Omron CX-Programmer project NewProject (CX-Programmer 9.66)

# PLC LQK19011ICM: CP1H XA
I/O table (CPU CP1H-XA40DR-A): rack 0 slot 0 CJ1W-SCU21

## Global symbols (name address type ; comment)
AI_SAW_CURRENT 200 CHANNEL  ; ANALOG.INPUT1.SAW.CURRENT
AO_TRANS_VEL_REF 210 CHANNEL  ; TRANSVERSE.AXIS.VELOCITY.ANALOG.REFERENCE
0 CHANNEL  ; Zero Jog reference value first
0.04 BOOL  ; SPARE
0.05 BOOL  ; SPARE
1.01 BOOL  ; Spare
1.03 BOOL  ; Spare
D10 CHANNEL  ; Jog Velocity Reference Value
D1000 CHANNEL  ; First Dtata address of block table
D2000 CHANNEL  ; First Data Word of slab table
D8 CHANNEL  ; Interim Jog Storage Wd
D9 CHANNEL  ; Interim Storage word for Jog
H10.11 BOOL  ; MC.LONG.AXIS
H10.12 BOOL  ; MC.LONG.AXIS
H10.13 BOOL  ; MC.LONG.AXIS
H12.07 BOOL  ; MC.TRANSVERSE.AXIS
H12.08 BOOL  ; MC.TRANSVERSE.AXIS
H12.11 BOOL  ; MC.TRANSVERSE.AXIS
H12.12 BOOL  ; MC.TRANSVERSE.AXiS
H12.13 BOOL  ; MC.TRANSVERSE.AXIS
T0000 BOOL  ; Step 0 Timer Done
T0001 BOOL  ; Step 1 Timer Done
T0002 BOOL  ; Step 2 timer done
T0003 BOOL  ; Increment Slab Pulse Timer
T0004 BOOL  ; Slab Decrement Pulse Timer
T0005 BOOL  ; Block Increment Pulse Timer
T0006 BOOL  ; Block Decrement Pulse Timer
T0010 BOOL  ; Block Step 0 Timer
T0011 BOOL  ; Block Step 1 Timer
T0012 BOOL  ; Block Step 2 Timer
T0013 BOOL  ; Block Step 3 Timer
T0014 BOOL  ; Block Step 4 timer
T0015 BOOL  ; Block Step 5 Timer
T0016 BOOL  ; Block Step 6 Timer
W121.02 BOOL  ; Previous Block
W121.03 BOOL  ; Previous Slab of Current Block
W121.04 BOOL  ; Next Slab of current Block
W121.05 BOOL  ; Next Block Select
W121.06 BOOL  ; Write Current Block to Storage (HMI PB)
W121.07 BOOL  ; Clear Data
W12.00 BOOL  ; Slab Change Data Storage and Display Update Step 0
W12.01 BOOL  ; Step 1
W12.02 BOOL  ; Step 2
W12.03 BOOL  ; Step 3
W12.04 BOOL  ; Step 4
W12.05 BOOL  ; Step 5
W12.06 BOOL  ; Step 6
W12.15 BOOL  ; Loop Step Reset
W13.00 BOOL  ; Step 0 in Progress
W13.01 BOOL  ; Step 1 in Progress
W13.02 BOOL  ; Step 2 in Progress
W13.03 BOOL  ; Step 3 in Progress
W13.04 BOOL  ; Step 4 in Progress
W13.05 BOOL  ; Step 5 in Progress
W13.06 BOOL  ; Step 6 in Progress
W14.00 BOOL  ; Step 0 Done
W14.01 BOOL  ; Step 1 Done
W14.02 BOOL  ; Step 2 Done
W14.03 BOOL  ; Step 3 Done
W14.04 BOOL  ; Step 4 Done
W14.05 BOOL  ; Step 5 Done
W14.06 BOOL  ; Step 6 Done
W150 CHANNEL  ; Block Number Captured
W151 CHANNEL  ; Number of Words for Blocks
W152 CHANNEL  ; Slab Count Work Word for Block Pointer
W153 CHANNEL  ; Offset Calculate for Last Slab Count
W154 CHANNEL  ; Offset Mid Calc
W156 CHANNEL  ; Offset Calc'd
W158 CHANNEL  ; Slab Record Offset Interim
W15.00 BOOL  ; Block Change Data Storage and Display Update Step 0
W15.01 BOOL  ; Loop Step 1
W15.02 BOOL  ; Loop Step 2
W15.03 BOOL  ; Loop Step 3
W15.04 BOOL  ; Loop Step 4
W15.05 BOOL  ; Loop Step 5
W15.06 BOOL  ; Loop Step 6
W15.15 BOOL  ; Loop Step Reset
W160 CHANNEL  ; Slab Offset Result
W16.00 BOOL  ; Step 0 in Progress
W16.01 BOOL  ; Loop Step 1 in Progress
W16.02 BOOL  ; Loop Step 2 in Progress
W16.03 BOOL  ; Loop Step 3 in Progress
W16.04 BOOL  ; Loop Step 4 in Progress
W16.05 BOOL  ; Loop Step 5 in Progress
W16.06 BOOL  ; Loop Step 6 in Progress
W16.10 BOOL  ; Slab Data Read in Progress
W16.11 BOOL  ; Block Data Read in Progress
W17.00 BOOL  ; Step 0 Done
W17.01 BOOL  ; Loop Step 1 Done
W17.02 BOOL  ; Loop Step 2 Complete
W17.03 BOOL  ; Loop Sstep 3 Complete
W17.04 BOOL  ; Loop Step 4 Complete
W17.05 BOOL  ; Loop Step 5 Complete
W17.06 BOOL  ; Loop Step 6 Complete
W190 CHANNEL  ; Slab Pointer Offset Adjustment
W191 CHANNEL  ; Block 1 Slab Count Capture
W192 CHANNEL  ; Slab Offset Addition for This Block
W193 CHANNEL  ; Slab_ID_Raw
W194 CHANNEL  ; Slab Pointer Calculated
W195 CHANNEL  ; Slab Offset Previous
W196 CHANNEL  ; Slab_Offset_Constant_Calculated
W197 CHANNEL  ; Block_Selected_Base
W198 CHANNEL  ; Block Pointer Offset Calculated
W19.00 BOOL  ; Test Bit
W19.01 BOOL  ; Self Toggle
W200 CHANNEL  ; Block ID
W201 CHANNEL  ; Number Of Blocks
W202 CHANNEL  ; Current Block Height
W203 CHANNEL  ; Current Block Start Edge
W204 CHANNEL  ; Current Block Length
W205 CHANNEL  ; Current Block First Cut Location
W206 CHANNEL  ; Current Block SLab Count
W207 CHANNEL  ; Slab ID
W208 CHANNEL  ; Current Slab Size in inches
W209 CHANNEL  ; Current Slab Quantity to cut
W20.00 BOOL  ; Block Incremented Pulse - Lead
W20.01 BOOL  ; Block Decremented Pulse - Lead
W20.02 BOOL  ; Slab Incremented Pulse - Lead
W20.03 BOOL  ; Slab Decremented Pulse - Lead
W20.04 BOOL  ; Slab Count Capture Trap
W20.05 BOOL  ; Block Read In Progress
W20.06 BOOL  ; Slab Count Changed from Block Read
W20.07 BOOL  ; Slab Pointer Updating
W20.08 BOOL  ; Update Working Offset
W20.09 BOOL  ; Block Pointer Calculate Enable
W20.10 BOOL  ; Increment Block Pointer
W20.11 BOOL  ; Decrement Block Pointer
W20.12 BOOL  ; First_Pass_Read
W20.14 BOOL  ; Block Offset Calculated
W20.15 BOOL  ; Block Program Control Enabled
W21.00 BOOL  ; Blade Kerf Data Write to Storage
W21.01 BOOL  ; Blade Kerf Read from Storage
W21.02 BOOL  ; Cut Depth Write to Storage
W21.03 BOOL  ; Cut Depth Read from Storage
W21.04 BOOL  ; Target Saw Current in Amps Write to Storage
W21.05 BOOL  ; Target Saw Current in Amps Read from Storage
W21.06 BOOL  ; Read Slab Data from Storage
W21.07 BOOL  ; Block Data Write to Storage
W21.08 BOOL  ; Automatic Number of Blocks Update
W21.09 BOOL  ; Slab Pointer Control Enabled
W21.10 BOOL  ; Increment Slab Offset
W21.11 BOOL  ; Decrement Slab Offset
W21.12 BOOL  ; Automatic Number of Slabs Update
W21.13 BOOL  ; Slab Pointer Reset
W21.14 BOOL  ; Block Pointer Reset
W22.00 BOOL  ; Slab Pointer Calculated
W22.01 BOOL  ; Block Pointer Changed
W22.02 BOOL  ; Current Block Selected Changed Initiate Block Data Write
W22.03 BOOL  ; Block Data Write Step Zero Complete
W22.04 BOOL  ; Block Data Write Complete
W22.05 BOOL  ; Capture Current Slab Words
W22.06 BOOL  ; Slab Data Write In Progress
W22.07 BOOL  ; Slab Data Write Complete
W22.08 BOOL  ; Block Offset Adjusted
W22.09 BOOL  ; Block Offset Adjust Complete
W22.10 BOOL  ; Block Data Read in Progress
W22.11 BOOL  ; Block Data Read >
W22.12 BOOL  ; Block Data Read Complete
W22.13 BOOL  ; Slab Offset Adjust in Progress
W22.14 BOOL  ; Slab Offset Adjust >
W22.15 BOOL  ; Slab Offset Adjust Complete
W23.00 BOOL  ; Slab Offset Init
W23.01 BOOL  ; Slab Offset Pointer Updating
W23.02 BOOL  ; Slab Offset Updated
W23.03 BOOL  ; Slab Data Read in Progress
W23.04 BOOL  ; Slab Data Read >
W23.05 BOOL  ; Slab Data Read Complete
W23.15 BOOL  ; Slab Offset Init Complete
W24.01 BOOL  ; Offset Init Step 1 Complete
W24.02 BOOL  ; OffsetInit Step 2 Complete
W24.03 BOOL  ; Offset Init Step 3 Complete
W250 CHANNEL  ; Offset value for Second word in indirect addressed storage area for Block Start Edge
W251 CHANNEL  ; Offset Value for Third word in Storge area for block length
W252 CHANNEL  ; Offset value calculated for 4th word in Storage area for block First Cut
W253 CHANNEL  ; Offset value calculated for number of slabs for current block
W256 CHANNEL  ; Last Slab Count from First Block
W257 CHANNEL  ; Offset adjust
W25.01 BOOL  ; Offset Init Step 1 In Progress
W25.02 BOOL  ; Offset Init Step 2 In Progress
W25.03 BOOL  ; Offset Init Step 3 In Progress
W26.00 BOOL  ; Minus Slab Offset Init
W26.01 BOOL  ; Minus Offset Init Step 1
W26.02 BOOL  ; Minus Offset Init Step 2
W26.03 BOOL  ; Minus Offset Init Step 3
W26.15 BOOL  ; Minus Slab Offset Init Complete
W27.01 BOOL  ; Minus Offset Init Step 1 Complete
W27.02 BOOL  ; Minus Offset Init Step 2 Complete
W27.03 BOOL  ; Minus Offset Init Step 3 Complete
W28.01 BOOL  ; Minus Offset Init Step 1 In Progress
W28.02 BOOL  ; Minus Offset Init Step 2 In Progress
W28.03 BOOL  ; Minus Offset Init Step 3 In Progress
W300 CHANNEL  ; Blade Kerf Working
W301 CHANNEL  ; Cut Depth Working
W302 CHANNEL  ; Target Current Working
W30.00 BOOL  ; OI.MESSAGE.INTERNAL.TRIGGER.MSG0
W30.01 BOOL  ; OI.MESSAGE.INTERNAL.TRIGGER.MSG1
W312 CHANNEL  ; Last Height Value for Current Block
W313 CHANNEL  ; Current Block Stored Height Data
W314 CHANNEL  ; Curren Block Last Start Edge
W315 CHANNEL  ; Current Block Stored Start Edge
W316 CHANNEL  ; Current Block Last Length
W317 CHANNEL  ; Current Block Stored Length
W318 CHANNEL  ; Current Block Last First Cut Position
W319 CHANNEL  ; Current Block Stored First Cut Location
W320 CHANNEL  ; Current Block Last Number of Slabs
W321 CHANNEL  ; Current Block Stored Slab Count
W322 CHANNEL  ; Current Slab Last Width
W323 CHANNEL  ; Current Slab Stored Width
W324 CHANNEL  ; Current Slab Last Quantity
W325 CHANNEL  ; Current Slab Stored Quantity
W37.00 BOOL  ; Current Height and Last Height are not Equal after Block Inc/Dec
W37.01 BOOL  ; Last Height and Stored Height are not Equal
W37.02 BOOL  ; Current Block Start Edge and Last Block Start Edge are Not Equal
W37.03 BOOL  ; Last Block Start Edge and Stored Value are Not Equal
W37.04 BOOL  ; Current Block Length and Last Block Length are Not Equal
W37.05 BOOL  ; Last Block Length and Stored Length are Not Equal
W37.06 BOOL  ; Current and Last First Cut Location are Not Equal
W37.07 BOOL  ; Last and Stored First Cut Location are Not Equal
W37.08 BOOL  ; Last and Current Slab Count are Not Equal
W37.09 BOOL  ; Last and Stored Slab Count are Not Equal
W37.10 BOOL  ; Current and Last Slab Size are Not Equal
W37.11 BOOL  ; Last and Stored Slab Sizes are Not Equal
W37.12 BOOL  ; Last and Current Slab Qty are Not Equal
W37.13 BOOL  ; Last and Stored Slab Qty are Not Equal
W400 CHANNEL  ; Temporary Storage for Block Data Used in Slab Offset Calc
W400.00 BOOL  ; Data Write Step
W400.01 BOOL  ; Data Offset Adjust Step
W400.02 BOOL  ; Data Read Step
W400.03 BOOL  ; End Step
W404 CHANNEL  ; # of Slabs for current Block
W405 CHANNEL  ; Number of words used by slabs in this block
W406 CHANNEL  ; Temporary Offset Storage word
W40.00 BOOL  ; Data Write/Read Sequence Initiate
W40.01 BOOL  ; Data Write Step Action
W40.02 BOOL  ; Data Offset Adjust Action
W40.03 BOOL  ; Data Read Step Action
W41.00 BOOL  ; Slab Data Write in Progress
W41.01 BOOL  ; Slab Data Write >
W41.02 BOOL  ; Slab Offset Adjust in Progress
W41.03 BOOL  ; Calulating Number of Words to Read
W90.00 BOOL  ; Block Data Write Step 0
W90.01 BOOL  ; Slab Data Write Step 1
W90.02 BOOL  ; Change Block Offset Pointer
W90.03 BOOL  ; Read Block Data
W90.04 BOOL  ; Slab Offset Adjust
W90.05 BOOL  ; Slab Offset Pointer Update
W90.06 BOOL  ; Slab Data Read
W90.07 BOOL  ; Last Step
BLADE_KERF D210 CHANNEL  ; BLADE.KERF.VALUE
BLK_DATA_END_ADR D1999 CHANNEL  ; Block Datat Tabe dimension end
BLK_DATA_STRT_ADR D1000 CHANNEL  ; Dimension the Block Data Table
BLK_DAT_RD_INIT H90.01 BOOL  ; Block Data Read Initiated
BLK_DAT_WRT_INIT H90.00 BOOL  ; Block Data Write Initiated
Block_Pointer Calculate_Pointer
CUT_DEPTH D211 CHANNEL  ; CUT.DEPTH.VALUE.PROGRAMMED
CUT_TRGT_CUR D212 CHANNEL  ; CUT.TARGET.CURRENT
DI_ENC_0_A 0.08 BOOL  ; ENCODER.0.A
DI_ENC_0_B 0.09 BOOL  ; ENCODER.0.B
DI_ENC_0_Z 0.03 BOOL  ; ENCODER.0.Z
DI_ENC_1_A 0.06 BOOL  ; ENCODER.1.A
DI_ENC_1_B 0.07 BOOL  ; ENCODER.1.B
DI_ENC_1_Z 0.02 BOOL  ; ENCODER.1.Z
DI_FLOW_SW 1.00 BOOL  ; WATER.FLOW.SWITCH
DI_LONG_MASTER_DRV_OK 0.10 BOOL  ; IO.LONG.AXIS.MASTER.DRIVE.OKAY.INPUT
DI_LONG_SLAVE_DRV_OK 0.01 BOOL  ; IO.LONG.SLAVE.DRIVE.OKAY.INPUT
DI_MCR_ON 0.00 BOOL  ; MCR.ON.POWER.ON
DI_SAFETY_ITLK 1.02 BOOL  ; SAFETY.GATE.INTERLOCK.INPUT
DI_SFT_STRT_FLT 0.11 BOOL  ; SAW.SOFT.START.FAULT
DI_TRANS_AXIS_DRV_OK 1.04 BOOL  ; IO.TRANSVERSE.AXIS.DRIVE.OKAY.INPUT
DI_TRANS_FWD 1.06 BOOL  ; TRANSVERSE.AXIS.FORWARD.LIMT.PROXIMITY
DI_TRANS_HOME 1.05 BOOL  ; TRANSVERSE.AXIS.HOME.PROXIMITY
DI_VERT_AXIS_DRV_OK 1.10 BOOL  ; IO.VERTICAL.AXIS.DRIVE.OKAY.INPUT
DI_VERT_FWD 1.08 BOOL  ; VERTICAL.AXIS.FORWARD.LIMIT
DI_VERT_HOME 1.07 BOOL  ; VERTICAL.AXIS.HOME.PROXIMITY
DO_ALARM_ANNUN 101.01 BOOL  ; ALARM.ANNUNCIATOR
DO_LAZER_ON 101.07 BOOL  ; LASER.ON
DO_LONG_AXIS_DRV_INDEX_CMD 101.02 BOOL  ; LONG.AXIS.MASTER.DRV.INDEX.COMMAND
DO_LONG_AXIS_HOME_INIT 101.06 BOOL  ; LONG.AXIS.MASTER.DRV.INITIATE.HOME.MOVE
DO_LONG_AXIS_JOG_LEFT 101.04 BOOL  ; LONG.AXIS.MASTER.DRV.JOG.LEFT
DO_LONG_AXIS_JOG_RIGHT 101.05 BOOL  ; LONG.AXIS.MASTER.DRV.JOG.RIGHT
DO_SFT_STRT_RUN 100.01 BOOL  ; SOFT.START.RUN
DO_SFT_STRT_STP 101.00 BOOL  ; SOFT.START.STOP
DO_TRANS_AXIS_FWD 100.04 BOOL  ; TRANSVERSE.AXIS.FORWARD
DO_TRANS_AXIS_REV 100.05 BOOL  ; TRANSVERSE.AXIS.REVERSE
DO_VERT_AXIS_BRK 101.03 BOOL  ; VERTICAL.AXIS.BRAKE
DO_VERT_AXIS_LWR 100.03 BOOL  ; VERTICAL.AXIS.LOWER
DO_VERT_AXIS_RAISE 100.02 BOOL  ; VERTICAL.AXIS.RAISE
DO_VERT_AXIS_SPD_SEL 100.06 BOOL  ; VERTICAL.AXIS.SPEED.SELECT
DO_WATER_VLV 100.00 BOOL  ; WATER.VALVE
GLOBAL_HOME_REQUEST W0.15 BOOL  ; GLOBAL.HOME.REQUEST
HSC0_Init HSC0_INIT
HSC0_PWR_INIT H0.00 BOOL  ; HSC.0.PWR.INIT
HSC1_Init HSC1_INIT
HSC1_PWR_INIT H0.01 BOOL  ; HSC.1.PWR.INIT
IO_LAZER_PWR_OK H15.00 BOOL  ; IO.LAZER.POWER.OKAY
IO_LAZER_SG_OK H15.01 BOOL  ; IO.LAZER.SAFETY.GATE.OKAY
IO_SAW_NOT_SAFE_TO_RUN H13.03 BOOL  ; IO.SAW.NOT.SAFE.TO.RUN
IO_SAW_PWR_OK H13.00 BOOL  ; IO.SAW.POWER.OKAY
IO_SAW_SAFE_TO_RUN H13.02 BOOL  ; IO.SAW.SAFE.TO.RUN
IO_SAW_SG_OK H13.01 BOOL  ; IO.SAW.SAFETY.GATE.OKAY
IO_Saw_Safe_To_Run Op_2_State
IO_WTR_PWR_OK H14.00 BOOL  ; IO.WATER.POWER.OKAY
IO_WTR_SG_OK H14.01 BOOL  ; IO.WATER.SAFETY.GATE.OKAY
LAXISMFDBK A276 CHANNEL  ; LONG.AXIS.MASTER.FEEDBACK
MAIN_PWR_ERR W0.05 BOOL  ; MAIN.POWER.ERR
MC_AXIS_LONG_FDBK D5000 CHANNEL  ; Axis Actual Position Feedback from Drive
MC_Axis_Long_Home MC_Axis_Home
MC_LONG_AXIS_AUTO_NOK H10.03 BOOL  ; MC.LONG.AXIS.AUTO.NOT.OKAY
MC_LONG_AXIS_AUTO_OK H10.02 BOOL  ; MC.LONG.AXIS.AUTO.OKAY
MC_LONG_AXIS_DRV_ACT 302.00 BOOL  ; MC.LONG.AXIS.DRIVE.ACTIVE
MC_LONG_AXIS_DRV_AT_ZERO 303.00 BOOL  ; MC.LONG.AXIS.DRIVE.AT.ZERO.SPEED
MC_LONG_AXIS_DRV_ERR H10.05 BOOL  ; MC.LONG.AXIS.DRIVE.ERROR
MC_LONG_AXIS_DRV_JOG_REF D5005 INT  ; MC.LONG.AXIS.DRIVE.JOG.SPEED.REFERENCE
MC_LONG_AXIS_DRV_MAINS_LOSS 315.00 BOOL  ; MC.LONG.AXIS.MAINS.LOSS.FAULT
MC_LONG_AXIS_DRV_OK 301.00 BOOL  ; MC.LONG.AXIS.DRIVE.OKAY
MC_LONG_AXIS_DRV_OKAY H10.04 BOOL  ; MC.LONG.AXIS.DRIVE.OKAY
MC_LONG_AXIS_DRV_OL 317.00 BOOL  ; MC.LONG.AXIS.DRIVE.OVERLOAD.FAULT
MC_LONG_AXIS_DRV_RST 333.00 BOOL  ; MC.LONG.AXIS.DRIVE.RESET
MC_LONG_AXIS_DRV_UV 316.00 BOOL  ; MC.LONG.AXIS.DRIVE.BUS.UNDER.VOLTAGE.ERROR
MC_LONG_AXIS_DRV_WRN 319.00 BOOL  ; MC.LONG.AXIS.DRIVE.WARNING.[FAULT EXISTS]
MC_LONG_AXIS_ERR H10.14 BOOL  ; LONG.AXIS.ERROR.EXISTS
MC_LONG_AXIS_GATE_OK H10.01 BOOL  ; LONG.AXIS.SAFETY.GATE.OKAY
MC_LONG_AXIS_HOME_CMD_INT H10.08 BOOL  ; MC.LONG.AXIS.HOME.COMMAND.INTERNAL
MC_LONG_AXIS_HOM_DN H10.09 BOOL  ; MC.LONG.AXIS.HOME.DONE
MC_LONG_AXIS_JOGL_CMD H10.06 BOOL  ; MC.LONG.AXIS.JOG.LEFT.COMMAND
MC_LONG_AXIS_JOGR_CMD H10.07 BOOL  ; MC.LONG.AXIS.JOG.RIGHT.COMMAND
MC_LONG_AXIS_JOG_ERR H10.10 BOOL  ; MC.LONG.AXIS.JOG.ERROR
MC_LONG_AXIS_POS_REF_CMD D4 CHANNEL  ; MC.LONG.AXIS.POSITION.REFERENCE.COMMAND.VALUE
MC_LONG_AXIS_PWR_OK H10.00 BOOL  ; LONG.AXIS.POWER.OKAY
MC_LONG_AXIS_RDY H10.15 BOOL  ; LONG.AXIS.MOTION.READY
MC_LONG_AXIS_TEMP_FLT 318.00 BOOL  ; MC.LONG.AXIS.DRIVE.OVER.TEMPERATURE.FAULT
MC_Long_Axis_Drv_OK Op_2_State
MC_Long_Axis_Jog_Cmd MC_Axis_Jog
MC_Op_Trans_Axis_Jog_Cmd MC_Axis_Jog
MC_PERM_TRANS_AXIS_AUTO_NOK H12.03 BOOL  ; MC.PERMISSIVE.TRANSVERSE.AXIS.AUTO.NOK
MC_PERM_TRANS_AXIS_AUTO_OK H12.02 BOOL  ; MC.PERMISSIVE.TRANSVERSE.AXIS.AUTO.OK
MC_TRANS_AXIS_DRV_ACT 402.00 BOOL  ; MC.TRANSVERSE.AXIS.DRIVE.ACTIVE
MC_TRANS_AXIS_DRV_AT_ZERO_SPD 403.00 BOOL  ; MC.TRANSVERSE.AXIS.DRIVE.AT.ZERO.SPEED
MC_TRANS_AXIS_DRV_ERR H12.05 BOOL  ; MC.TRANSVERSE.AXIS.DRIVE.ERROR
MC_TRANS_AXIS_DRV_GNRL_ERR 419.00 BOOL  ; MC.TRANSVERSE.AXIS.DRIVE.GENERAL.ERROR
MC_TRANS_AXIS_DRV_JOG_REF D6005 INT  ; MC.TRANSVERSE.AXIS.DRIVE.JOG.REFERENCE.IN.HZ.REAL
MC_TRANS_AXIS_DRV_MAINS_LOSS 415.00 BOOL  ; MC.TRANSVERSE.AXIS.DRIVE.MAINS.LOSS
MC_TRANS_AXIS_DRV_NOT_STOP 410.00 BOOL  ; MC.TRANSVERSE.AXIS.DRIVE.NOT.STOP
MC_TRANS_AXIS_DRV_OK 401.00 BOOL  ; MC.TRANSVERSE.AXIS.DRIVE.OKAY.STATUS
MC_TRANS_AXIS_DRV_OK_PERM H12.04 BOOL  ; MC.PERMISSIVE.TRANSVERSE.AXIS.DRIVE.OKAY
MC_TRANS_AXIS_DRV_OL 417.00 BOOL  ; MC.TRANSVERSE.AXIS.DRIVE.OVERLOAD.ERROR
MC_TRANS_AXIS_DRV_PREC_REF_COARSE D6010 INT  ; MC.TRANSVERSE.AXIS.DRIVE.PRECISION.REFERENCE.COARSE.VALUE
MC_TRANS_AXIS_DRV_PREC_REF_FINE D6012 INT  ; MC.TRANSVERSE.AXIS.DRIVE.PRECISION.REFERENCE.FINE.VALUE
MC_TRANS_AXIS_DRV_PREC_REF_SEL 444.00 BOOL  ; MC.TRANSVERSE.AXIS.DRIVE.PRECISION.REFERENCE.SELECT
MC_TRANS_AXIS_DRV_RESET 433.00 BOOL  ; MC.TRANSVERSE.AXIS.DRIVE.ERROR.RESET
MC_TRANS_AXIS_DRV_RUN_FWD 405.00 BOOL  ; MC.TRANSVERSE.AXIS.DRIVE.RUN.FORWARD
MC_TRANS_AXIS_DRV_RUN_REV 407.00 BOOL  ; MC.TRANSVERSE.AXIS.DRIVE.RUN.REVERSE
MC_TRANS_AXIS_DRV_TEMP_ERR 418.00 BOOL  ; MC.TRANSVERSE.AXIS.DRIVE.TEMPERATURE.ERROR
MC_TRANS_AXIS_ERR H12.14 BOOL  ; TRANSVERSE.AXIS.ERROR.EXISTS
MC_TRANS_AXIS_JOG_ACT H12.09 BOOL  ; MC.TRANSVERSE.AXIS.JOG.COMMAND.ACTIVE
MC_TRANS_AXIS_JOG_CMD_ERR H12.10 BOOL  ; MC.TRANSVERSE.AXIS.JOG.COMMAND.ERROR
MC_TRANS_AXIS_JOG_EN H12.06 BOOL  ; MC.TRANSVERSE.AXIS.JOG.ENABLED
MC_TRANS_AXIS_JOG_FWD 406.00 BOOL  ; MC.TRANSVERSE.AXIS.DRIVE.JOG.FORWARD
MC_TRANS_AXIS_JOG_REV 408.00 BOOL  ; MC.TRANSVERSE.AXIS.DRIVE.JOG.REVERSE
MC_TRANS_AXIS_PWR_OK H12.00 BOOL  ; TRANSVERSE.AXIS.POWER.OKAY
MC_TRANS_AXIS_READY H12.15 BOOL  ; MC.TRANSVERSE.READY
MC_TRANS_AXIS_SAFETY_GATE_OK H12.01 BOOL  ; TRANSVERSE.AXIS.SAFETY.GATE.OKAY
MC_TRAN_AXIS_DRV_EN 404.00 BOOL  ; MC.TRANSVERSE.AXIS.DRIVE.ENABLE
MC_VERT_AXISDRV_NOT_STP 510.00 BOOL  ; MC.VERTICAL.AXIS.DRIVE.NOT.STOP
MC_VERT_AXIS_AUTO_NOK H11.03 BOOL  ; MC.VERTTICAL.AXIS.AUTO.NOK
MC_VERT_AXIS_AUTO_OK H11.02 BOOL  ; MC.VERTICAL.AXIS.AUTO.OK
MC_VERT_AXIS_CMD_LWR H11.05 BOOL  ; MC_VERT_AXIS_CMD_LOWER
MC_VERT_AXIS_CMD_RAISE H11.04 BOOL  ; MC_VERT_AXIS_CMD_RAISE
MC_VERT_AXIS_DRV_ACT 502.00 BOOL  ; MC.VERTICAL.AXIS.DRIVE.ACTIVE
MC_VERT_AXIS_DRV_AT_ZERO_SPD 503.00 BOOL  ; MC.VERTICAL.AXIS.DRIVE.AT.ZERO.SPEED
MC_VERT_AXIS_DRV_EN 504.00 BOOL  ; MC.VERTICAL.AXIS.DRIVE.ENABLE
MC_VERT_AXIS_DRV_GNRL_ERR 519.00 BOOL  ; MC.VERTICAL.AXIS.DRIVE.GENERAL.ERROR
MC_VERT_AXIS_DRV_MAINS_LOSS 515.00 BOOL  ; MC.VERTICAL.AXIS.DRIVE.MAINS.LOSS
MC_VERT_AXIS_DRV_OK 501.00 BOOL  ; MC.VERTICAL.AXIS.DRIVE.OKAY
MC_VERT_AXIS_DRV_OL 517.00 BOOL  ; MC.VERTICAL.AXIS.DRIVE.OVERLOAD.ERROR
MC_VERT_AXIS_DRV_PREC_REF_SEL 544.00 BOOL  ; MC.VERTICAL.AXIS.DRIVE.PRECISION.REFERENCE.SELECT
MC_VERT_AXIS_DRV_RESET 533.00 BOOL  ; MC.VERTICAL.AXIS.DRIVE.RESET
MC_VERT_AXIS_DRV_RUN_REV 507.00 BOOL  ; MC.VERTICAL.AXIS.DRIVE.RUN.REVERSE
MC_VERT_AXIS_DRV_TEMP_ERR 518.00 BOOL  ; MC.VERTICAL.AXIS.DRIVE.TEMPERATURE.ERROR
MC_VERT_AXIS_ERR H11.14 BOOL  ; MC.VERTICAL.AXIS.ERROR
MC_VERT_AXIS_JOG_FWD 506.00 BOOL  ; MC.VERTICAL.AXIS.DRIVE.JOG.FORWARD
MC_VERT_AXIS_JOG_REV 508.00 BOOL  ; MC.VERTICAL.AXIS.JOG.REVERSE
MC_VERT_AXIS_PWR_OK H11.00 BOOL  ; VERTICAL.AXIS.POWER.OKAY
MC_VERT_AXIS_RDY H11.15 BOOL  ; MC.VERTICAL.AXIS.READY
MC_VERT_AXIS_RUN_FWD 505.00 BOOL  ; MC.VERTICAL.AXIS.DRIVE.RUN.FORWARD
MC_VERT_AXIS_SAFETY_GATE_OK H11.01 BOOL  ; VERTICAL.AXIS.SAFETY.GATE.OKAY
MODE_AUTO_IND W130.14 BOOL  ; AUTOMATIC.MODE.INDICATOR
MODE_MAN_IND W130.13 BOOL  ; MANUAL.MODE.INDICATOR
MODE_SEL_AUTO W0.09 BOOL  ; MODE.SELECT.AUTOMATIC
MODE_SEL_AUTO_EN W0.11 BOOL  ; MODE.SELECT.AUTO.MODE.ENABLED
MODE_SEL_EN W0.07 BOOL  ; MODE.SELECT.ENABLED
MODE_SEL_MAN W0.08 BOOL  ; MODE.SELECT.MANUAL
MODE_SEL_MAN_EN W0.10 BOOL  ; MODE.SELECT.MANUAL.MODE.ENABLED
Mode_Select Op_Mode_Sel
OI_ALM_CLR W111 WORD  ; OI.ALARM.MESSAGE.COLOUR
OI_ALM_SEL W110 WORD  ; OI.ALARM.MESSAGE.SELECT
OI_CTL_WORD_1 W120 WORD  ; OI.CONTROL.WORD.1
OI_CTL_WORD_2 W121 WORD  ; OI.CONTROL.WORD.2
OI_CTRL_CYCLE_START W120.02 BOOL  ; OI.CONTROL.AUTOMATIC.CYCLE.START.PB
OI_CTRL_CYCLE_STOP_PB W120.01 BOOL  ; OI.CONTROL.AUTOMATIC.CYCLE.STOP.PB
OI_CTRL_H_A_SEL W120.00 BOOL  ; OI.CONTROL.HAND.AUTO.SELECTOR
OI_CTRL_MAC_STOP W120.03 BOOL  ; OI.CONTROL.AUTOMATIC.CYCLE.MACHINE.STOP
OI_HOME_ALL_PB W120.04 BOOL  ; OI.HOME.ALL.PB
OI_IND_WORD_1 W130 WORD  ; OI.INDICATE.WORD.1
OI_IND_WORD_2 W131 WORD  ; OI.INDICATE.WORD.2
OI_LONG_AXIS_JOG_MINUS W120.15 BOOL  ; OI.LONG.AXIS.JOG.MINUS.PB
OI_LONG_AXIS_JOG_PLUS W121.00 BOOL  ; OI.LONG.AXIS.JOG.PLUS.PB
OI_MSG_CLR W101 INT  ; OI.MESSAGE.COLOUR
OI_MSG_SEL W100 INT  ; OI.MESSAGE.SELECT
OI_SAW_STP_PB W120.08 BOOL  ; OI.SAW.STOP.PB
OI_SAW_STRT_PB W120.07 BOOL  ; OI.SAW.START.PB
OI_TRANS_AXIS_JOG_HOME_PB W120.13 BOOL  ; OI.TRANSVERSE.AXIS.JOG.HOME.PB
OI_TRANS_AXIS_JO_FWD_PB W120.14 BOOL  ; OI.TRANSVERSE.AXIS.JOG.FORWARD.PB
OI_VERT_AXIS_JOG_FWD_PB W120.11 BOOL  ; OI.VERTICAL.AXIS.JOG.FORWARD.PB
OI_VERT_AXIS_JOG_HOME_PB W120.10 BOOL  ; OI.VERTICAL.AXIS.JOG.HOME.PB
OI_WTR_ON_SEL W120.06 BOOL  ; OI.WATER.ON.SELECTOR
OOI_LAZER_ON_SEL W120.05 BOOL  ; OI.LAZER.ON.SELECTOR
OP_FIRST_CYC_CMPLT H0.02 BOOL  ; FIRST.CYCLE.COMPLETED
OP_Power_On_Check Op_2_State
Op_Gate_Monitor Op_2_State
Op_Long_Axis_Mode Op_Mode_Sel
Op_Mode_Ind Mode_Ind
Op_Mode_Indication Mode_Ind
Op_Perm_Long_Auto Op_2_State
Op_Trans_Auto_Ok Op_2_State
Op_Trans_Axis_Drv_Ok Op_2_State
Op_Vert_Auto_Ok Op_2_State
POWER_ON W0.03 BOOL  ; POWER.ON.MAIN
SAFETY_GATE_ERR W0.06 BOOL  ; SAFETY.GATE.ERR
SAFETY_GATE_OK W0.04 BOOL  ; SAFETY.GATE.OKAY
SLAB_DATA_END_ADR D2999 CHANNEL  ; DIMENSION.SLAB.DATA.TABLE.END
SLAB_DATA_START_ADR D2000 CHANNEL  ; DIMENSION.SLAB.DATA.TABLE.START
Slab_Pointer Calculate_Pointer
TRANS_POS_FDBK A272 CHANNEL  ; TRANSVERSE.POSITION.FEEDBACK.RAW
VERT_POS_FDBK A270 CHANNEL  ; VERTICAL.POSITION.FEEDBACK.RAW

## Program Main (cyclic task 0)
; Main saw program file
Local symbols
Channel_for_HSC0 INT  ; The Default Channel for HSC 0
EW195 CHANNEL
HSC0_Init_Plx W0.00 BOOL  ; HSC0 Initialised at Power Up
HSC1_Init_Plx W1.00 BOOL  ; HSC1 Initialised at power up
Long_Axis_En_Request BOOL
POWER_ON_ERR BOOL

### Section Init_HSC

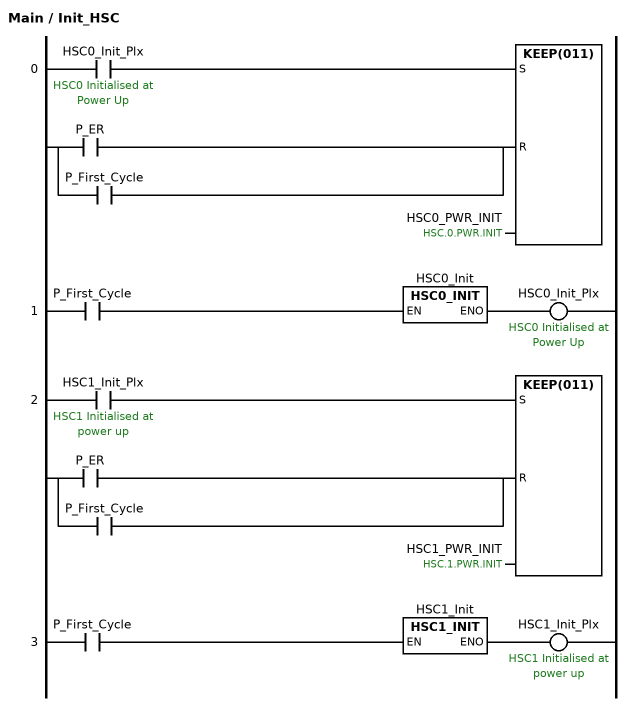
; rung 0
LD HSC0_Init_Plx  ; HSC0 Initialised at Power Up
LD P_ER
OR P_First_Cycle
KEEP(011) HSC0_PWR_INIT  ; HSC.0.PWR.INIT
; rung 1
LD P_First_Cycle
CALL HSC0_Init : HSC0_INIT ()
OUT HSC0_Init_Plx  ; HSC0 Initialised at Power Up
; rung 2
LD HSC1_Init_Plx  ; HSC1 Initialised at power up
LD P_ER
OR P_First_Cycle
KEEP(011) HSC1_PWR_INIT  ; HSC.1.PWR.INIT
; rung 3
LD P_First_Cycle
CALL HSC1_Init : HSC1_INIT ()
OUT HSC1_Init_Plx  ; HSC1 Initialised at power up

### Section Interlock_Alarm

### Section Ctl_Power

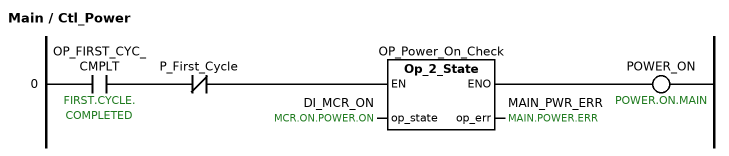
; rung 0
LD OP_FIRST_CYC_CMPLT  ; FIRST.CYCLE.COMPLETED
ANDNOT P_First_Cycle
CALL OP_Power_On_Check : Op_2_State (op_state := DI_MCR_ON, op_err => MAIN_PWR_ERR)  ; MCR.ON.POWER.ON, MAIN.POWER.ERR
OUT POWER_ON  ; POWER.ON.MAIN

### Section Ctl_Safety

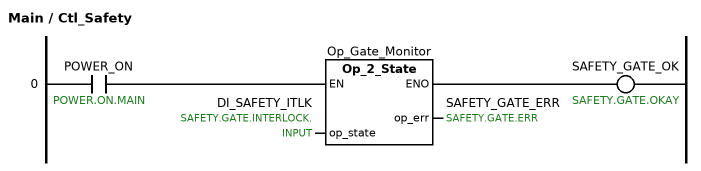
; rung 0
LD POWER_ON  ; POWER.ON.MAIN
CALL Op_Gate_Monitor : Op_2_State (op_state := DI_SAFETY_ITLK, op_err => SAFETY_GATE_ERR)  ; SAFETY.GATE.INTERLOCK.INPUT, SAFETY.GATE.ERR
OUT SAFETY_GATE_OK  ; SAFETY.GATE.OKAY

### Section Ctl_Mode

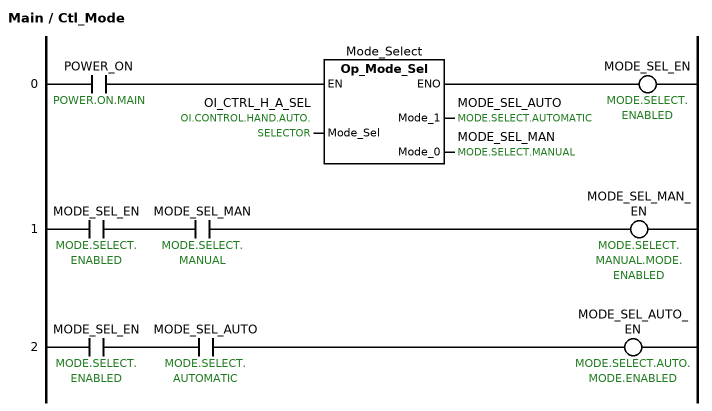
; rung 0
LD POWER_ON  ; POWER.ON.MAIN
CALL Mode_Select : Op_Mode_Sel (Mode_Sel := OI_CTRL_H_A_SEL, Mode_1 => MODE_SEL_AUTO, Mode_0 => MODE_SEL_MAN)  ; OI.CONTROL.HAND.AUTO.SELECTOR, MODE.SELECT.AUTOMATIC, MODE.SELECT.MANUAL
OUT MODE_SEL_EN  ; MODE.SELECT.ENABLED
; rung 1
LD MODE_SEL_EN  ; MODE.SELECT.ENABLED
AND MODE_SEL_MAN  ; MODE.SELECT.MANUAL
OUT MODE_SEL_MAN_EN  ; MODE.SELECT.MANUAL.MODE.ENABLED
; rung 2
LD MODE_SEL_EN  ; MODE.SELECT.ENABLED
AND MODE_SEL_AUTO  ; MODE.SELECT.AUTOMATIC
OUT MODE_SEL_AUTO_EN  ; MODE.SELECT.AUTO.MODE.ENABLED

### Section Ctl_Cycle_Start

### Section Ctl_Cycle_Stop

### Section Ctl_Home

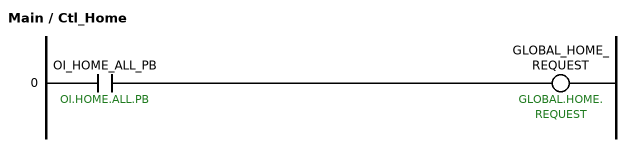
; rung 0
LD OI_HOME_ALL_PB  ; OI.HOME.ALL.PB
OUT GLOBAL_HOME_REQUEST  ; GLOBAL.HOME.REQUEST

### Section Ctl_Long_Axis

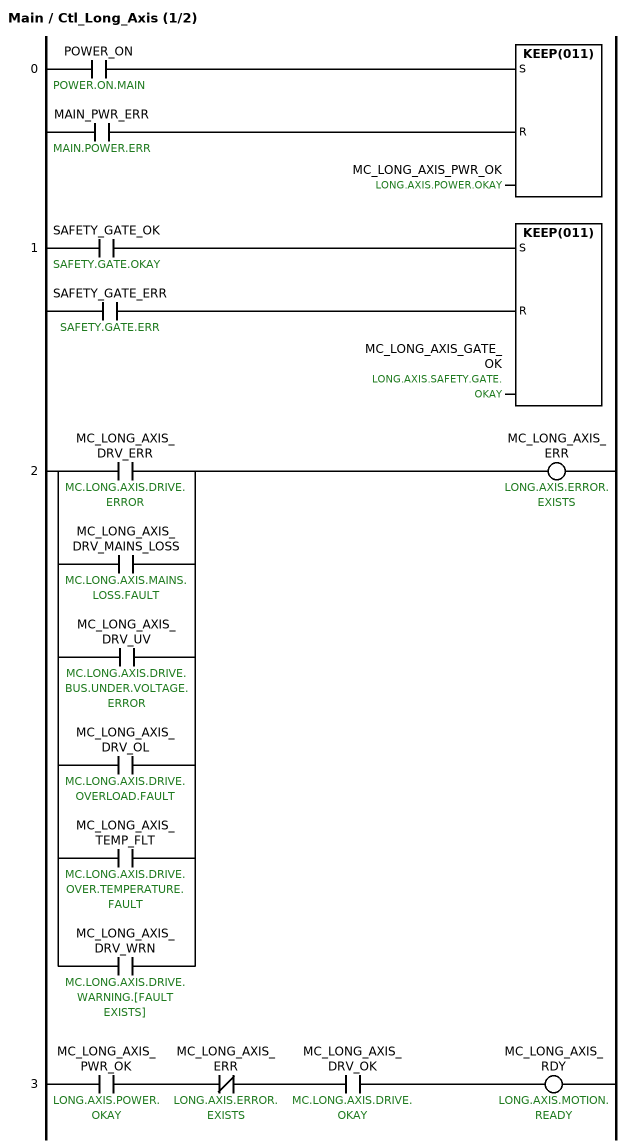
; rung 0
LD POWER_ON  ; POWER.ON.MAIN
LD MAIN_PWR_ERR  ; MAIN.POWER.ERR
KEEP(011) MC_LONG_AXIS_PWR_OK  ; LONG.AXIS.POWER.OKAY
; rung 1
LD SAFETY_GATE_OK  ; SAFETY.GATE.OKAY
LD SAFETY_GATE_ERR  ; SAFETY.GATE.ERR
KEEP(011) MC_LONG_AXIS_GATE_OK  ; LONG.AXIS.SAFETY.GATE.OKAY
; rung 2
LD MC_LONG_AXIS_DRV_ERR  ; MC.LONG.AXIS.DRIVE.ERROR
OR MC_LONG_AXIS_DRV_MAINS_LOSS  ; MC.LONG.AXIS.MAINS.LOSS.FAULT
OR MC_LONG_AXIS_DRV_UV  ; MC.LONG.AXIS.DRIVE.BUS.UNDER.VOLTAGE.ERROR
OR MC_LONG_AXIS_DRV_OL  ; MC.LONG.AXIS.DRIVE.OVERLOAD.FAULT
OR MC_LONG_AXIS_TEMP_FLT  ; MC.LONG.AXIS.DRIVE.OVER.TEMPERATURE.FAULT
OR MC_LONG_AXIS_DRV_WRN  ; MC.LONG.AXIS.DRIVE.WARNING.[FAULT EXISTS]
OUT MC_LONG_AXIS_ERR  ; LONG.AXIS.ERROR.EXISTS
; rung 3
LD MC_LONG_AXIS_PWR_OK  ; LONG.AXIS.POWER.OKAY
ANDNOT MC_LONG_AXIS_ERR  ; LONG.AXIS.ERROR.EXISTS
AND MC_LONG_AXIS_DRV_OK  ; MC.LONG.AXIS.DRIVE.OKAY
OUT MC_LONG_AXIS_RDY  ; LONG.AXIS.MOTION.READY

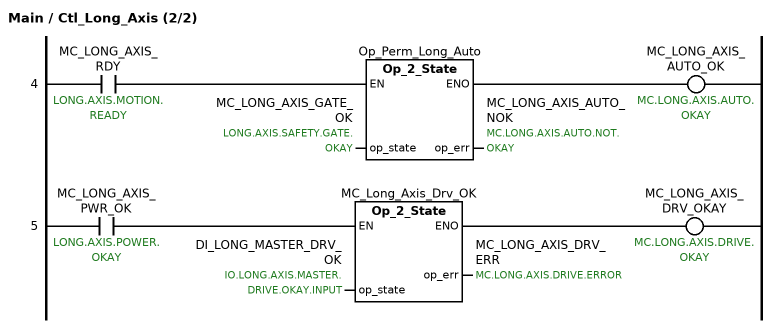
; rung 4
LD MC_LONG_AXIS_RDY  ; LONG.AXIS.MOTION.READY
CALL Op_Perm_Long_Auto : Op_2_State (op_state := MC_LONG_AXIS_GATE_OK, op_err => MC_LONG_AXIS_AUTO_NOK)  ; LONG.AXIS.SAFETY.GATE.OKAY, MC.LONG.AXIS.AUTO.NOT.OKAY
OUT MC_LONG_AXIS_AUTO_OK  ; MC.LONG.AXIS.AUTO.OKAY
; rung 5
LD MC_LONG_AXIS_PWR_OK  ; LONG.AXIS.POWER.OKAY
CALL MC_Long_Axis_Drv_OK : Op_2_State (op_state := DI_LONG_MASTER_DRV_OK, op_err => MC_LONG_AXIS_DRV_ERR)  ; IO.LONG.AXIS.MASTER.DRIVE.OKAY.INPUT, MC.LONG.AXIS.DRIVE.ERROR
OUT MC_LONG_AXIS_DRV_OKAY  ; MC.LONG.AXIS.DRIVE.OKAY

### Section Ctl_Vertical_Axis

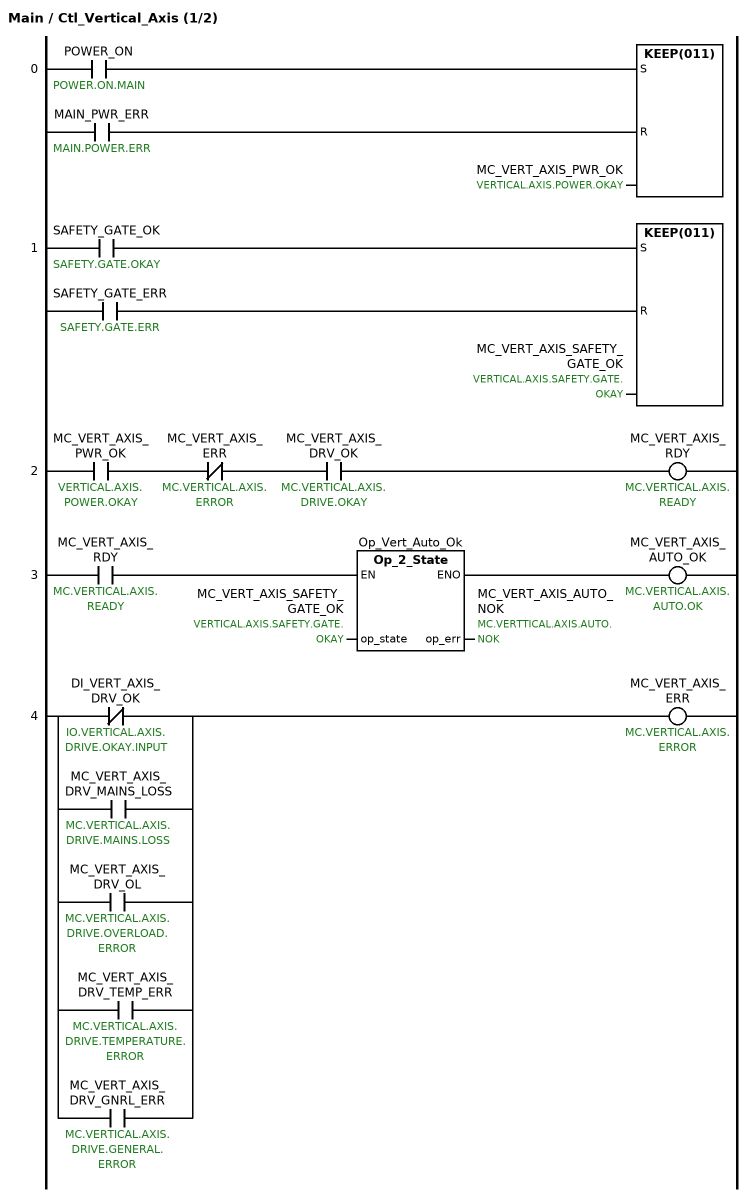
; rung 0
LD POWER_ON  ; POWER.ON.MAIN
LD MAIN_PWR_ERR  ; MAIN.POWER.ERR
KEEP(011) MC_VERT_AXIS_PWR_OK  ; VERTICAL.AXIS.POWER.OKAY
; rung 1
LD SAFETY_GATE_OK  ; SAFETY.GATE.OKAY
LD SAFETY_GATE_ERR  ; SAFETY.GATE.ERR
KEEP(011) MC_VERT_AXIS_SAFETY_GATE_OK  ; VERTICAL.AXIS.SAFETY.GATE.OKAY
; rung 2
LD MC_VERT_AXIS_PWR_OK  ; VERTICAL.AXIS.POWER.OKAY
ANDNOT MC_VERT_AXIS_ERR  ; MC.VERTICAL.AXIS.ERROR
AND MC_VERT_AXIS_DRV_OK  ; MC.VERTICAL.AXIS.DRIVE.OKAY
OUT MC_VERT_AXIS_RDY  ; MC.VERTICAL.AXIS.READY
; rung 3
LD MC_VERT_AXIS_RDY  ; MC.VERTICAL.AXIS.READY
CALL Op_Vert_Auto_Ok : Op_2_State (op_state := MC_VERT_AXIS_SAFETY_GATE_OK, op_err => MC_VERT_AXIS_AUTO_NOK)  ; VERTICAL.AXIS.SAFETY.GATE.OKAY, MC.VERTTICAL.AXIS.AUTO.NOK
OUT MC_VERT_AXIS_AUTO_OK  ; MC.VERTICAL.AXIS.AUTO.OK
; rung 4
LDNOT DI_VERT_AXIS_DRV_OK  ; IO.VERTICAL.AXIS.DRIVE.OKAY.INPUT
OR MC_VERT_AXIS_DRV_MAINS_LOSS  ; MC.VERTICAL.AXIS.DRIVE.MAINS.LOSS
OR MC_VERT_AXIS_DRV_OL  ; MC.VERTICAL.AXIS.DRIVE.OVERLOAD.ERROR
OR MC_VERT_AXIS_DRV_TEMP_ERR  ; MC.VERTICAL.AXIS.DRIVE.TEMPERATURE.ERROR
OR MC_VERT_AXIS_DRV_GNRL_ERR  ; MC.VERTICAL.AXIS.DRIVE.GENERAL.ERROR
OUT MC_VERT_AXIS_ERR  ; MC.VERTICAL.AXIS.ERROR

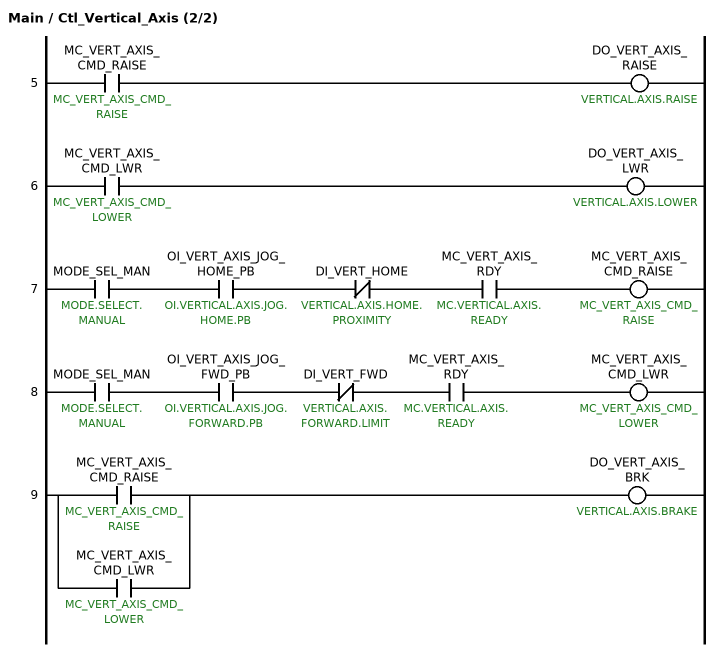
; rung 5
LD MC_VERT_AXIS_CMD_RAISE  ; MC_VERT_AXIS_CMD_RAISE
OUT DO_VERT_AXIS_RAISE  ; VERTICAL.AXIS.RAISE
; rung 6
LD MC_VERT_AXIS_CMD_LWR  ; MC_VERT_AXIS_CMD_LOWER
OUT DO_VERT_AXIS_LWR  ; VERTICAL.AXIS.LOWER
; rung 7
LD MODE_SEL_MAN  ; MODE.SELECT.MANUAL
AND OI_VERT_AXIS_JOG_HOME_PB  ; OI.VERTICAL.AXIS.JOG.HOME.PB
ANDNOT DI_VERT_HOME  ; VERTICAL.AXIS.HOME.PROXIMITY
AND MC_VERT_AXIS_RDY  ; MC.VERTICAL.AXIS.READY
OUT MC_VERT_AXIS_CMD_RAISE  ; MC_VERT_AXIS_CMD_RAISE
; rung 8
LD MODE_SEL_MAN  ; MODE.SELECT.MANUAL
AND OI_VERT_AXIS_JOG_FWD_PB  ; OI.VERTICAL.AXIS.JOG.FORWARD.PB
ANDNOT DI_VERT_FWD  ; VERTICAL.AXIS.FORWARD.LIMIT
AND MC_VERT_AXIS_RDY  ; MC.VERTICAL.AXIS.READY
OUT MC_VERT_AXIS_CMD_LWR  ; MC_VERT_AXIS_CMD_LOWER
; rung 9
LD MC_VERT_AXIS_CMD_RAISE  ; MC_VERT_AXIS_CMD_RAISE
OR MC_VERT_AXIS_CMD_LWR  ; MC_VERT_AXIS_CMD_LOWER
OUT DO_VERT_AXIS_BRK  ; VERTICAL.AXIS.BRAKE

### Section Ctl_Transverse_Axis

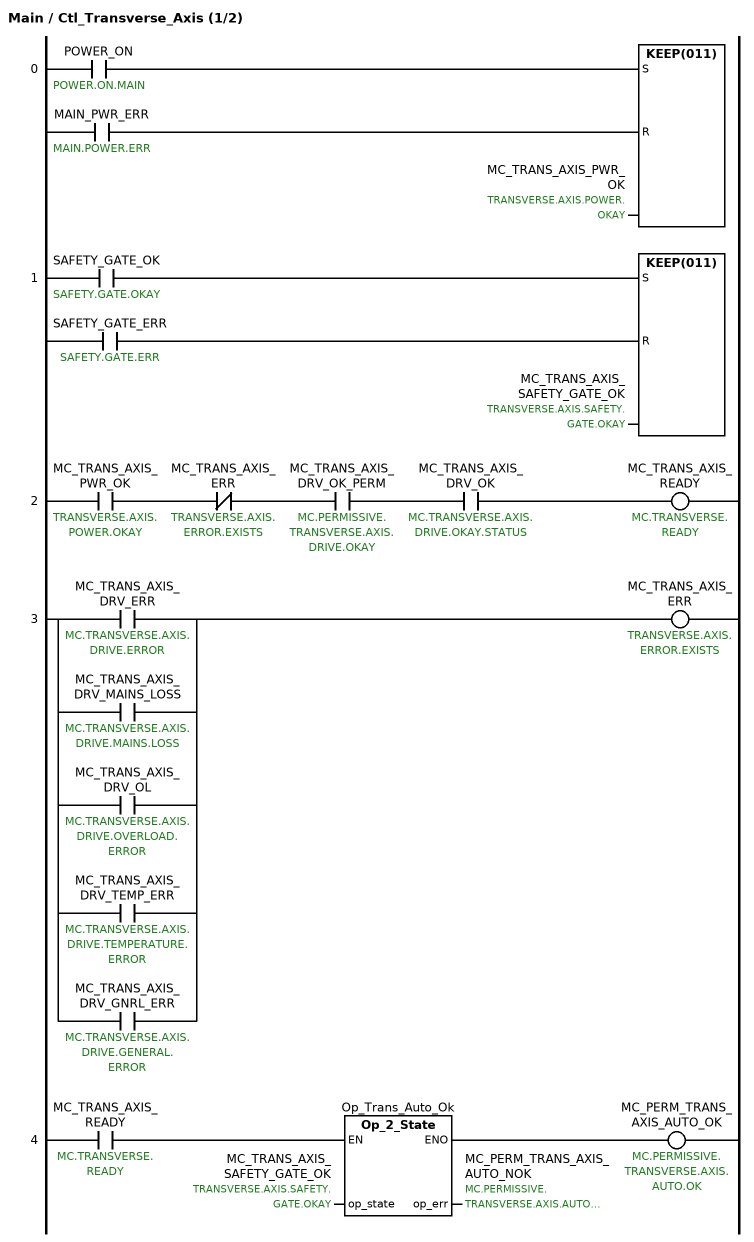
; rung 0
LD POWER_ON  ; POWER.ON.MAIN
LD MAIN_PWR_ERR  ; MAIN.POWER.ERR
KEEP(011) MC_TRANS_AXIS_PWR_OK  ; TRANSVERSE.AXIS.POWER.OKAY
; rung 1
LD SAFETY_GATE_OK  ; SAFETY.GATE.OKAY
LD SAFETY_GATE_ERR  ; SAFETY.GATE.ERR
KEEP(011) MC_TRANS_AXIS_SAFETY_GATE_OK  ; TRANSVERSE.AXIS.SAFETY.GATE.OKAY
; rung 2
LD MC_TRANS_AXIS_PWR_OK  ; TRANSVERSE.AXIS.POWER.OKAY
ANDNOT MC_TRANS_AXIS_ERR  ; TRANSVERSE.AXIS.ERROR.EXISTS
AND MC_TRANS_AXIS_DRV_OK_PERM  ; MC.PERMISSIVE.TRANSVERSE.AXIS.DRIVE.OKAY
AND MC_TRANS_AXIS_DRV_OK  ; MC.TRANSVERSE.AXIS.DRIVE.OKAY.STATUS
OUT MC_TRANS_AXIS_READY  ; MC.TRANSVERSE.READY
; rung 3
LD MC_TRANS_AXIS_DRV_ERR  ; MC.TRANSVERSE.AXIS.DRIVE.ERROR
OR MC_TRANS_AXIS_DRV_MAINS_LOSS  ; MC.TRANSVERSE.AXIS.DRIVE.MAINS.LOSS
OR MC_TRANS_AXIS_DRV_OL  ; MC.TRANSVERSE.AXIS.DRIVE.OVERLOAD.ERROR
OR MC_TRANS_AXIS_DRV_TEMP_ERR  ; MC.TRANSVERSE.AXIS.DRIVE.TEMPERATURE.ERROR
OR MC_TRANS_AXIS_DRV_GNRL_ERR  ; MC.TRANSVERSE.AXIS.DRIVE.GENERAL.ERROR
OUT MC_TRANS_AXIS_ERR  ; TRANSVERSE.AXIS.ERROR.EXISTS
; rung 4
LD MC_TRANS_AXIS_READY  ; MC.TRANSVERSE.READY
CALL Op_Trans_Auto_Ok : Op_2_State (op_state := MC_TRANS_AXIS_SAFETY_GATE_OK, op_err => MC_PERM_TRANS_AXIS_AUTO_NOK)  ; TRANSVERSE.AXIS.SAFETY.GATE.OKAY, MC.PERMISSIVE.TRANSVERSE.AXIS.AUTO.NOK
OUT MC_PERM_TRANS_AXIS_AUTO_OK  ; MC.PERMISSIVE.TRANSVERSE.AXIS.AUTO.OK

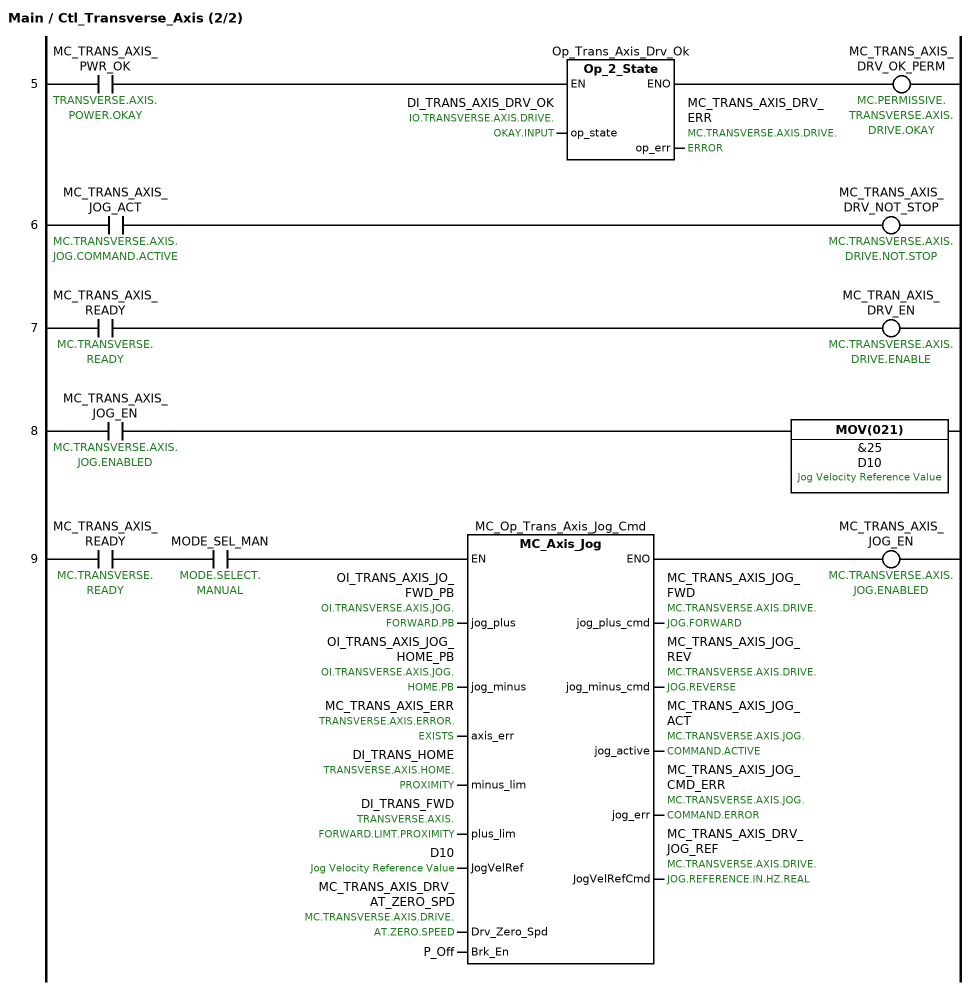
; rung 5
LD MC_TRANS_AXIS_PWR_OK  ; TRANSVERSE.AXIS.POWER.OKAY
CALL Op_Trans_Axis_Drv_Ok : Op_2_State (op_state := DI_TRANS_AXIS_DRV_OK, op_err => MC_TRANS_AXIS_DRV_ERR)  ; IO.TRANSVERSE.AXIS.DRIVE.OKAY.INPUT, MC.TRANSVERSE.AXIS.DRIVE.ERROR
OUT MC_TRANS_AXIS_DRV_OK_PERM  ; MC.PERMISSIVE.TRANSVERSE.AXIS.DRIVE.OKAY
; rung 6
LD MC_TRANS_AXIS_JOG_ACT  ; MC.TRANSVERSE.AXIS.JOG.COMMAND.ACTIVE
OUT MC_TRANS_AXIS_DRV_NOT_STOP  ; MC.TRANSVERSE.AXIS.DRIVE.NOT.STOP
; rung 7
LD MC_TRANS_AXIS_READY  ; MC.TRANSVERSE.READY
OUT MC_TRAN_AXIS_DRV_EN  ; MC.TRANSVERSE.AXIS.DRIVE.ENABLE
; rung 8
LD MC_TRANS_AXIS_JOG_EN  ; MC.TRANSVERSE.AXIS.JOG.ENABLED
MOV(021) &25 D10  ; Jog Velocity Reference Value
; rung 9
LD MC_TRANS_AXIS_READY  ; MC.TRANSVERSE.READY
AND MODE_SEL_MAN  ; MODE.SELECT.MANUAL
CALL MC_Op_Trans_Axis_Jog_Cmd : MC_Axis_Jog (jog_plus := OI_TRANS_AXIS_JO_FWD_PB, jog_minus := OI_TRANS_AXIS_JOG_HOME_PB, axis_err := MC_TRANS_AXIS_ERR, minus_lim := DI_TRANS_HOME, plus_lim := DI_TRANS_FWD, JogVelRef := D10, Drv_Zero_Spd := MC_TRANS_AXIS_DRV_AT_ZERO_SPD, Brk_En := P_Off, jog_plus_cmd => MC_TRANS_AXIS_JOG_FWD, jog_minus_cmd => MC_TRANS_AXIS_JOG_REV, jog_active => MC_TRANS_AXIS_JOG_ACT, jog_err => MC_TRANS_AXIS_JOG_CMD_ERR, JogVelRefCmd => MC_TRANS_AXIS_DRV_JOG_REF)  ; OI.TRANSVERSE.AXIS.JOG.FORWARD.PB, OI.TRANSVERSE.AXIS.JOG.HOME.PB, TRANSVERSE.AXIS.ERROR.EXISTS, TRANSVERSE.AXIS.HOME.PROXIMITY, TRANSVERSE.AXIS.FORWARD.LIMT.PROXIMITY, Jog Velocity Reference Value, MC.TRANSVERSE.AXIS.DRIVE.AT.ZERO.SPEED, MC.TRANSVERSE.AXIS.DRIVE.JOG.FORWARD, MC.TRANSVERSE.AXIS.DRIVE.JOG.REVERSE, MC.TRANSVERSE.AXIS.JOG.COMMAND.ACTIVE, MC.TRANSVERSE.AXIS.JOG.COMMAND.ERROR, MC.TRANSVERSE.AXIS.DRIVE.JOG.REFERENCE.IN.HZ.REAL
OUT MC_TRANS_AXIS_JOG_EN  ; MC.TRANSVERSE.AXIS.JOG.ENABLED

### Section Ctl_Saw

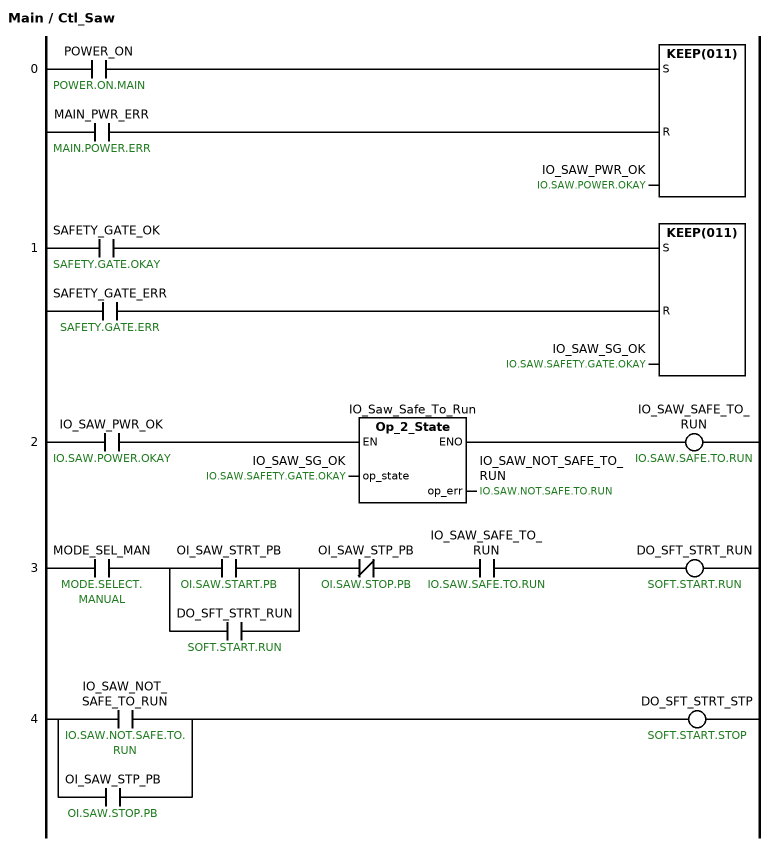
; rung 0
LD POWER_ON  ; POWER.ON.MAIN
LD MAIN_PWR_ERR  ; MAIN.POWER.ERR
KEEP(011) IO_SAW_PWR_OK  ; IO.SAW.POWER.OKAY
; rung 1
LD SAFETY_GATE_OK  ; SAFETY.GATE.OKAY
LD SAFETY_GATE_ERR  ; SAFETY.GATE.ERR
KEEP(011) IO_SAW_SG_OK  ; IO.SAW.SAFETY.GATE.OKAY
; rung 2
LD IO_SAW_PWR_OK  ; IO.SAW.POWER.OKAY
CALL IO_Saw_Safe_To_Run : Op_2_State (op_state := IO_SAW_SG_OK, op_err => IO_SAW_NOT_SAFE_TO_RUN)  ; IO.SAW.SAFETY.GATE.OKAY, IO.SAW.NOT.SAFE.TO.RUN
OUT IO_SAW_SAFE_TO_RUN  ; IO.SAW.SAFE.TO.RUN
; rung 3
LD MODE_SEL_MAN  ; MODE.SELECT.MANUAL
LD OI_SAW_STRT_PB  ; OI.SAW.START.PB
OR DO_SFT_STRT_RUN  ; SOFT.START.RUN
ANDLD
ANDNOT OI_SAW_STP_PB  ; OI.SAW.STOP.PB
AND IO_SAW_SAFE_TO_RUN  ; IO.SAW.SAFE.TO.RUN
OUT DO_SFT_STRT_RUN  ; SOFT.START.RUN
; rung 4
LD IO_SAW_NOT_SAFE_TO_RUN  ; IO.SAW.NOT.SAFE.TO.RUN
OR OI_SAW_STP_PB  ; OI.SAW.STOP.PB
OUT DO_SFT_STRT_STP  ; SOFT.START.STOP

### Section Ctl_Water

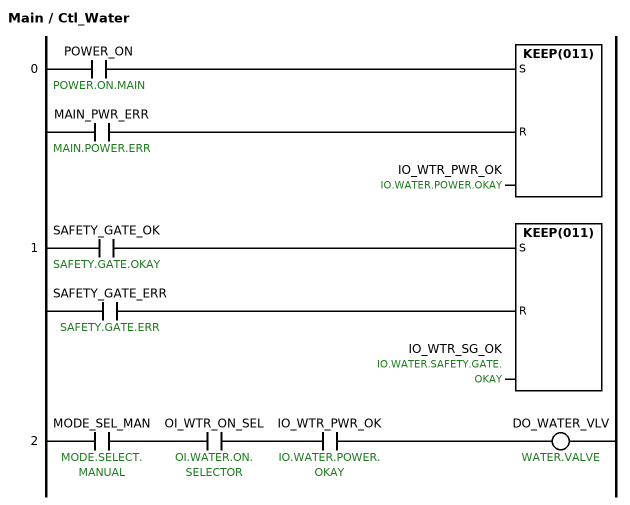
; rung 0
LD POWER_ON  ; POWER.ON.MAIN
LD MAIN_PWR_ERR  ; MAIN.POWER.ERR
KEEP(011) IO_WTR_PWR_OK  ; IO.WATER.POWER.OKAY
; rung 1
LD SAFETY_GATE_OK  ; SAFETY.GATE.OKAY
LD SAFETY_GATE_ERR  ; SAFETY.GATE.ERR
KEEP(011) IO_WTR_SG_OK  ; IO.WATER.SAFETY.GATE.OKAY
; rung 2
LD MODE_SEL_MAN  ; MODE.SELECT.MANUAL
AND OI_WTR_ON_SEL  ; OI.WATER.ON.SELECTOR
AND IO_WTR_PWR_OK  ; IO.WATER.POWER.OKAY
OUT DO_WATER_VLV  ; WATER.VALVE

### Section Ctl_Lazer

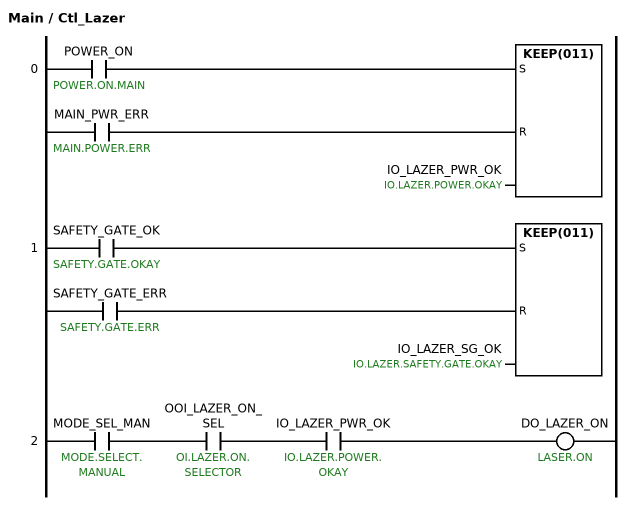
; rung 0
LD POWER_ON  ; POWER.ON.MAIN
LD MAIN_PWR_ERR  ; MAIN.POWER.ERR
KEEP(011) IO_LAZER_PWR_OK  ; IO.LAZER.POWER.OKAY
; rung 1
LD SAFETY_GATE_OK  ; SAFETY.GATE.OKAY
LD SAFETY_GATE_ERR  ; SAFETY.GATE.ERR
KEEP(011) IO_LAZER_SG_OK  ; IO.LAZER.SAFETY.GATE.OKAY
; rung 2
LD MODE_SEL_MAN  ; MODE.SELECT.MANUAL
AND OOI_LAZER_ON_SEL  ; OI.LAZER.ON.SELECTOR
AND IO_LAZER_PWR_OK  ; IO.LAZER.POWER.OKAY
OUT DO_LAZER_ON  ; LASER.ON

### Section Init_Recipe

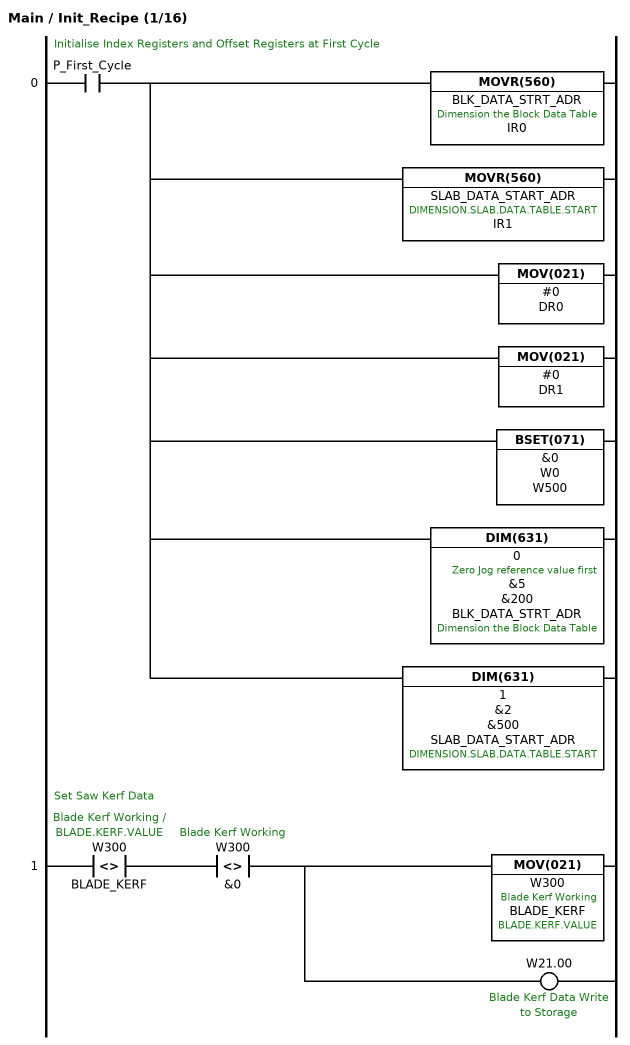
; rung 0: Initialise Index Registers and Offset Registers at First Cycle
LD P_First_Cycle
MOVR(560) BLK_DATA_STRT_ADR IR0  ; Dimension the Block Data Table
MOVR(560) SLAB_DATA_START_ADR IR1  ; DIMENSION.SLAB.DATA.TABLE.START
MOV(021) #0 DR0
MOV(021) #0 DR1
BSET(071) &0 W0 W500
DIM(631) 0 &5 &200 BLK_DATA_STRT_ADR  ; Zero Jog reference value first, Dimension the Block Data Table
DIM(631) 1 &2 &500 SLAB_DATA_START_ADR  ; DIMENSION.SLAB.DATA.TABLE.START
; rung 1: Set Saw Kerf Data
LD<>(305) W300 BLADE_KERF  ; Blade Kerf Working, BLADE.KERF.VALUE
AND<>(305) W300 &0  ; Blade Kerf Working
MOV(021) W300 BLADE_KERF  ; Blade Kerf Working, BLADE.KERF.VALUE
OUT W21.00  ; Blade Kerf Data Write to Storage

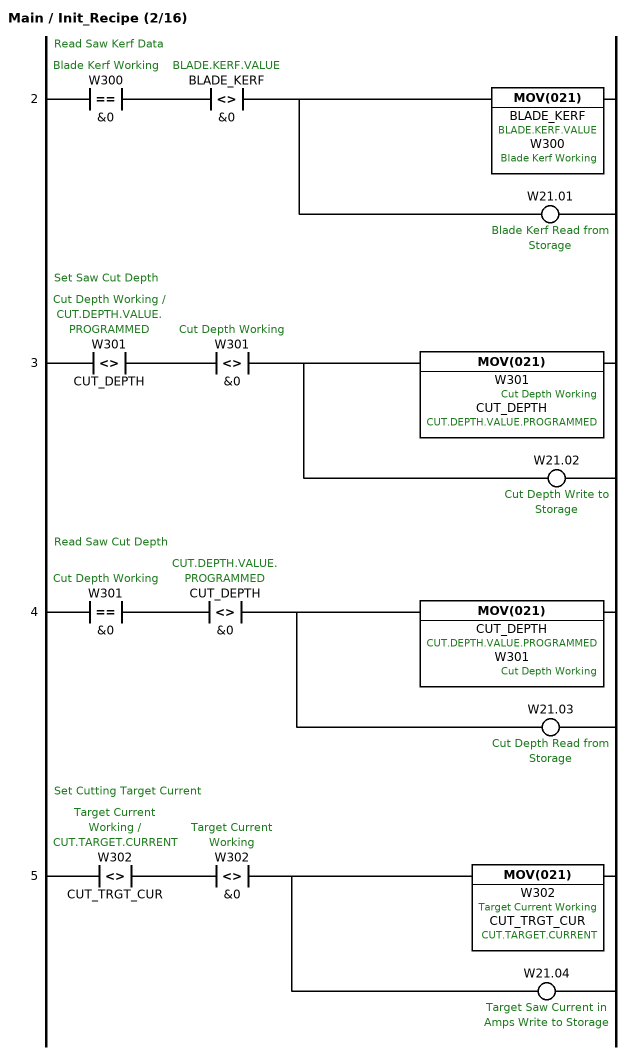
; rung 2: Read Saw Kerf Data
LD=(300) W300 &0  ; Blade Kerf Working
AND<>(305) BLADE_KERF &0  ; BLADE.KERF.VALUE
MOV(021) BLADE_KERF W300  ; BLADE.KERF.VALUE, Blade Kerf Working
OUT W21.01  ; Blade Kerf Read from Storage
; rung 3: Set Saw Cut Depth
LD<>(305) W301 CUT_DEPTH  ; Cut Depth Working, CUT.DEPTH.VALUE.PROGRAMMED
AND<>(305) W301 &0  ; Cut Depth Working
MOV(021) W301 CUT_DEPTH  ; Cut Depth Working, CUT.DEPTH.VALUE.PROGRAMMED
OUT W21.02  ; Cut Depth Write to Storage
; rung 4: Read Saw Cut Depth
LD=(300) W301 &0  ; Cut Depth Working
AND<>(305) CUT_DEPTH &0  ; CUT.DEPTH.VALUE.PROGRAMMED
MOV(021) CUT_DEPTH W301  ; CUT.DEPTH.VALUE.PROGRAMMED, Cut Depth Working
OUT W21.03  ; Cut Depth Read from Storage
; rung 5: Set Cutting Target Current
LD<>(305) W302 CUT_TRGT_CUR  ; Target Current Working, CUT.TARGET.CURRENT
AND<>(305) W302 &0  ; Target Current Working
MOV(021) W302 CUT_TRGT_CUR  ; Target Current Working, CUT.TARGET.CURRENT
OUT W21.04  ; Target Saw Current in Amps Write to Storage

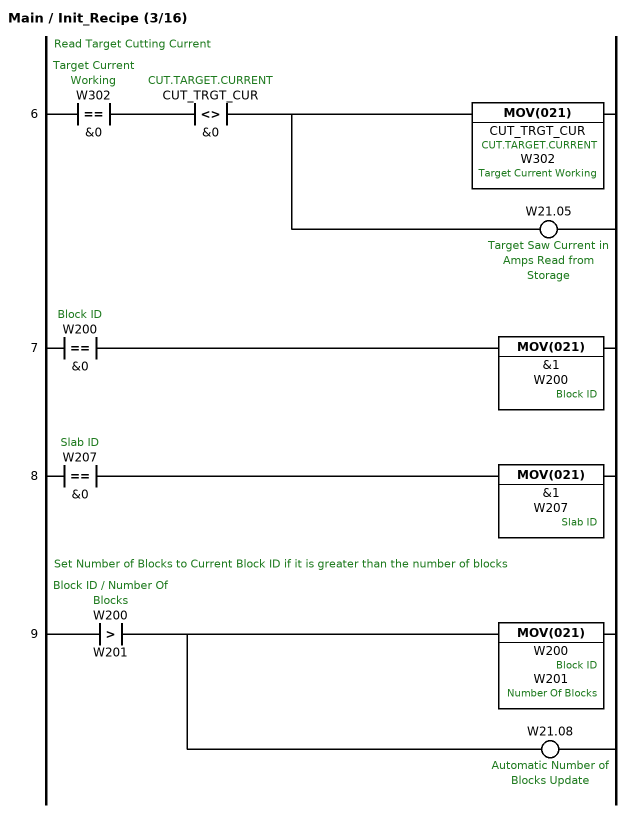
; rung 6: Read Target Cutting Current
LD=(300) W302 &0  ; Target Current Working
AND<>(305) CUT_TRGT_CUR &0  ; CUT.TARGET.CURRENT
MOV(021) CUT_TRGT_CUR W302  ; CUT.TARGET.CURRENT, Target Current Working
OUT W21.05  ; Target Saw Current in Amps Read from Storage
; rung 7
LD=(300) W200 &0  ; Block ID
MOV(021) &1 W200  ; Block ID
; rung 8
LD=(300) W207 &0  ; Slab ID
MOV(021) &1 W207  ; Slab ID
; rung 9: Set Number of Blocks to Current Block ID if it is greater than the number of blocks
LD>(320) W200 W201  ; Block ID, Number Of Blocks
MOV(021) W200 W201  ; Block ID, Number Of Blocks
OUT W21.08  ; Automatic Number of Blocks Update

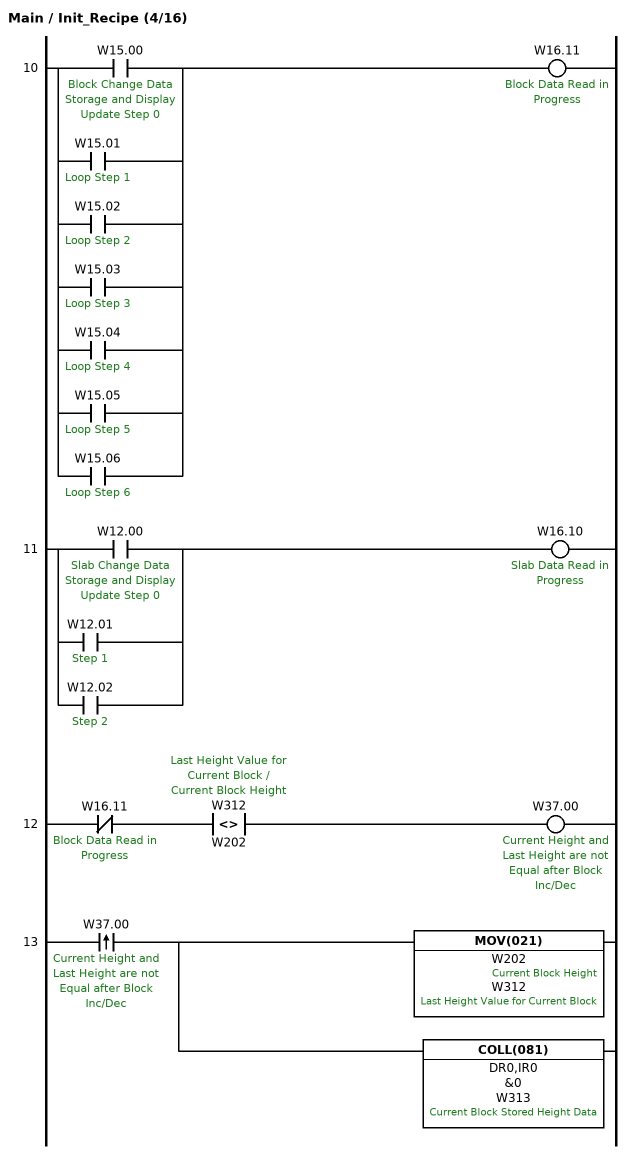
; rung 10
LD W15.00  ; Block Change Data Storage and Display Update Step 0
OR W15.01  ; Loop Step 1
OR W15.02  ; Loop Step 2
OR W15.03  ; Loop Step 3
OR W15.04  ; Loop Step 4
OR W15.05  ; Loop Step 5
OR W15.06  ; Loop Step 6
OUT W16.11  ; Block Data Read in Progress
; rung 11
LD W12.00  ; Slab Change Data Storage and Display Update Step 0
OR W12.01  ; Step 1
OR W12.02  ; Step 2
OUT W16.10  ; Slab Data Read in Progress
; rung 12
LDNOT W16.11  ; Block Data Read in Progress
AND<>(305) W312 W202  ; Last Height Value for Current Block, Current Block Height
OUT W37.00  ; Current Height and Last Height are not Equal after Block Inc/Dec
; rung 13
@LD W37.00  ; Current Height and Last Height are not Equal after Block Inc/Dec
MOV(021) W202 W312  ; Current Block Height, Last Height Value for Current Block
COLL(081) DR0,IR0 &0 W313  ; Current Block Stored Height Data

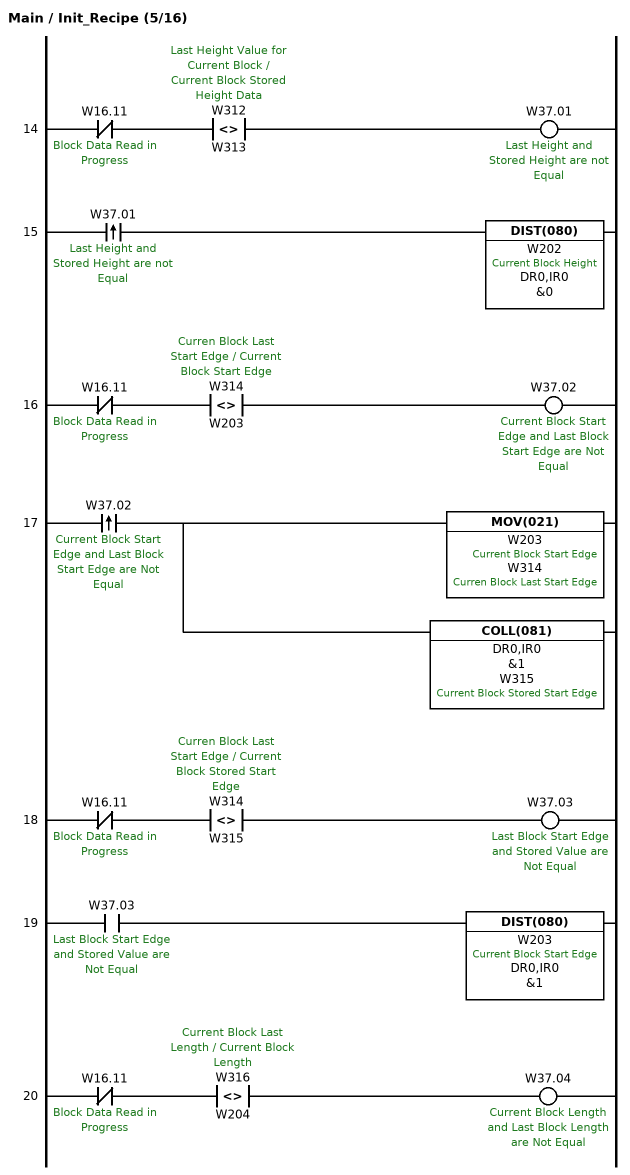
; rung 14
LDNOT W16.11  ; Block Data Read in Progress
AND<>(305) W312 W313  ; Last Height Value for Current Block, Current Block Stored Height Data
OUT W37.01  ; Last Height and Stored Height are not Equal
; rung 15
@LD W37.01  ; Last Height and Stored Height are not Equal
DIST(080) W202 DR0,IR0 &0  ; Current Block Height
; rung 16
LDNOT W16.11  ; Block Data Read in Progress
AND<>(305) W314 W203  ; Curren Block Last Start Edge, Current Block Start Edge
OUT W37.02  ; Current Block Start Edge and Last Block Start Edge are Not Equal
; rung 17
@LD W37.02  ; Current Block Start Edge and Last Block Start Edge are Not Equal
MOV(021) W203 W314  ; Current Block Start Edge, Curren Block Last Start Edge
COLL(081) DR0,IR0 &1 W315  ; Current Block Stored Start Edge
; rung 18
LDNOT W16.11  ; Block Data Read in Progress
AND<>(305) W314 W315  ; Curren Block Last Start Edge, Current Block Stored Start Edge
OUT W37.03  ; Last Block Start Edge and Stored Value are Not Equal
; rung 19
LD W37.03  ; Last Block Start Edge and Stored Value are Not Equal
DIST(080) W203 DR0,IR0 &1  ; Current Block Start Edge
; rung 20
LDNOT W16.11  ; Block Data Read in Progress
AND<>(305) W316 W204  ; Current Block Last Length, Current Block Length
OUT W37.04  ; Current Block Length and Last Block Length are Not Equal

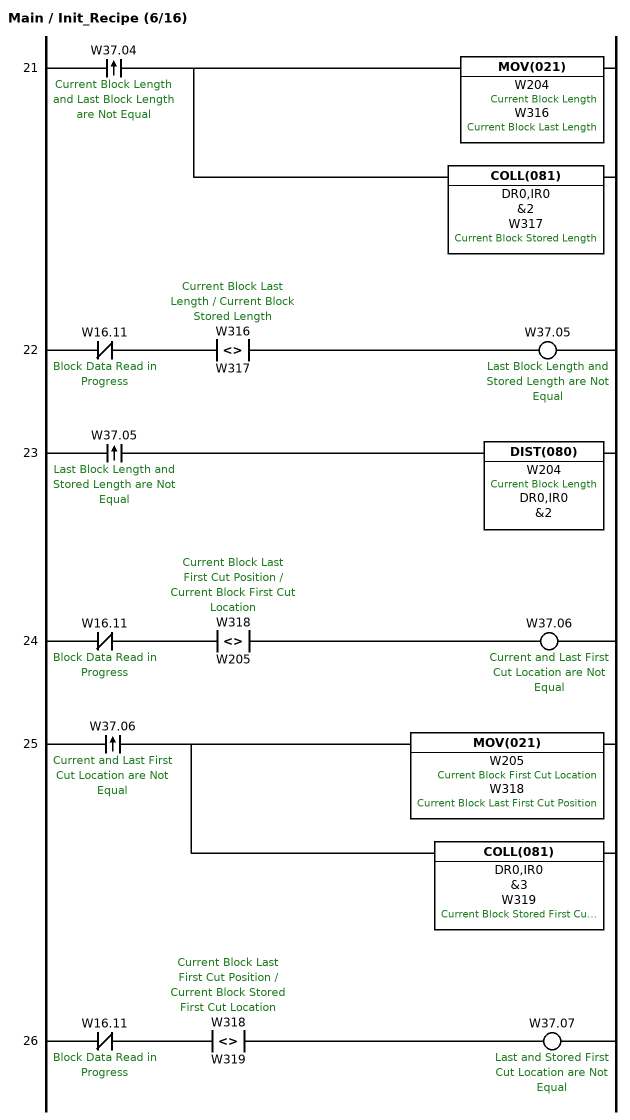
; rung 21
@LD W37.04  ; Current Block Length and Last Block Length are Not Equal
MOV(021) W204 W316  ; Current Block Length, Current Block Last Length
COLL(081) DR0,IR0 &2 W317  ; Current Block Stored Length
; rung 22
LDNOT W16.11  ; Block Data Read in Progress
AND<>(305) W316 W317  ; Current Block Last Length, Current Block Stored Length
OUT W37.05  ; Last Block Length and Stored Length are Not Equal
; rung 23
@LD W37.05  ; Last Block Length and Stored Length are Not Equal
DIST(080) W204 DR0,IR0 &2  ; Current Block Length
; rung 24
LDNOT W16.11  ; Block Data Read in Progress
AND<>(305) W318 W205  ; Current Block Last First Cut Position, Current Block First Cut Location
OUT W37.06  ; Current and Last First Cut Location are Not Equal
; rung 25
@LD W37.06  ; Current and Last First Cut Location are Not Equal
MOV(021) W205 W318  ; Current Block First Cut Location, Current Block Last First Cut Position
COLL(081) DR0,IR0 &3 W319  ; Current Block Stored First Cut Location
; rung 26
LDNOT W16.11  ; Block Data Read in Progress
AND<>(305) W318 W319  ; Current Block Last First Cut Position, Current Block Stored First Cut Location
OUT W37.07  ; Last and Stored First Cut Location are Not Equal

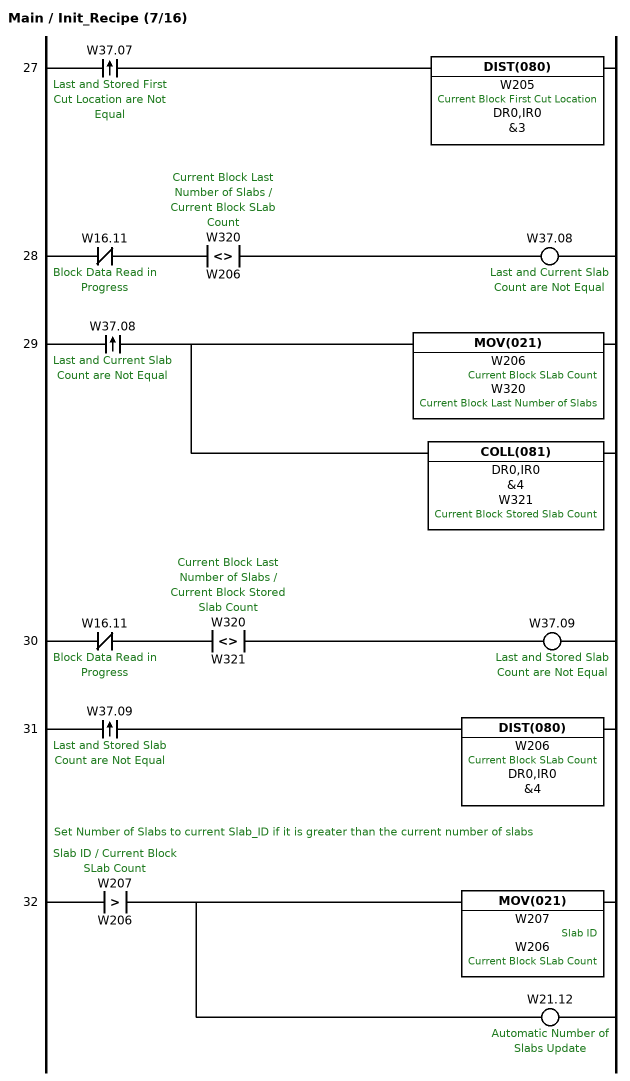
; rung 27
@LD W37.07  ; Last and Stored First Cut Location are Not Equal
DIST(080) W205 DR0,IR0 &3  ; Current Block First Cut Location
; rung 28
LDNOT W16.11  ; Block Data Read in Progress
AND<>(305) W320 W206  ; Current Block Last Number of Slabs, Current Block SLab Count
OUT W37.08  ; Last and Current Slab Count are Not Equal
; rung 29
@LD W37.08  ; Last and Current Slab Count are Not Equal
MOV(021) W206 W320  ; Current Block SLab Count, Current Block Last Number of Slabs
COLL(081) DR0,IR0 &4 W321  ; Current Block Stored Slab Count
; rung 30
LDNOT W16.11  ; Block Data Read in Progress
AND<>(305) W320 W321  ; Current Block Last Number of Slabs, Current Block Stored Slab Count
OUT W37.09  ; Last and Stored Slab Count are Not Equal
; rung 31
@LD W37.09  ; Last and Stored Slab Count are Not Equal
DIST(080) W206 DR0,IR0 &4  ; Current Block SLab Count
; rung 32: Set Number of Slabs to current Slab_ID if it is greater than the current number of slabs
LD>(320) W207 W206  ; Slab ID, Current Block SLab Count
MOV(021) W207 W206  ; Slab ID, Current Block SLab Count
OUT W21.12  ; Automatic Number of Slabs Update

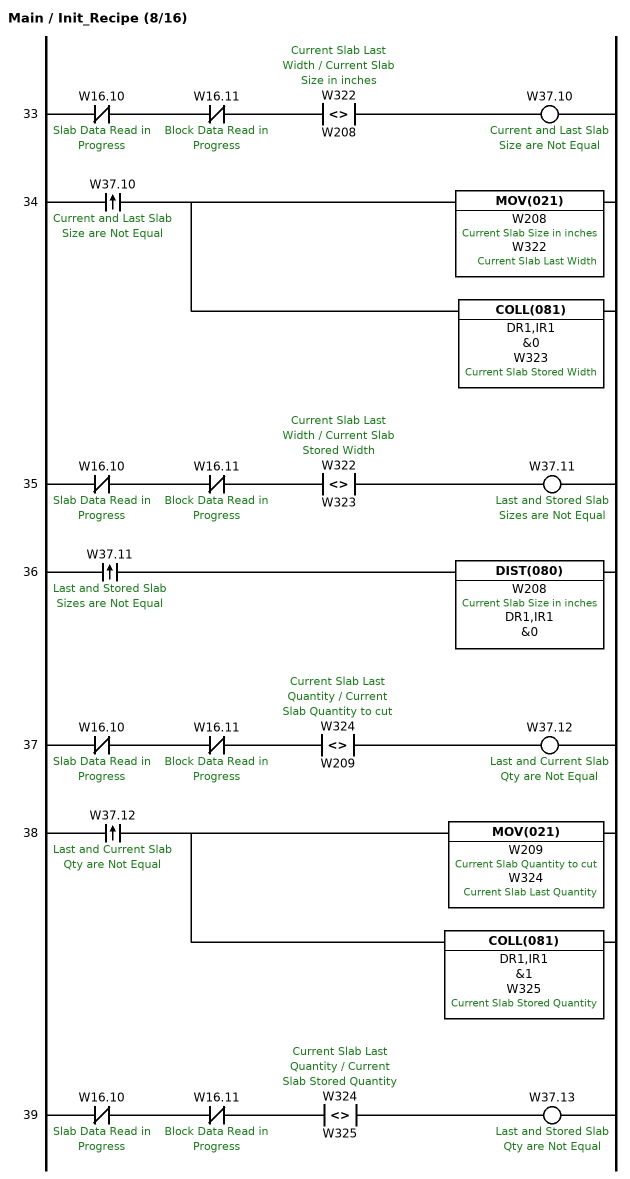
; rung 33
LDNOT W16.10  ; Slab Data Read in Progress
ANDNOT W16.11  ; Block Data Read in Progress
AND<>(305) W322 W208  ; Current Slab Last Width, Current Slab Size in inches
OUT W37.10  ; Current and Last Slab Size are Not Equal
; rung 34
@LD W37.10  ; Current and Last Slab Size are Not Equal
MOV(021) W208 W322  ; Current Slab Size in inches, Current Slab Last Width
COLL(081) DR1,IR1 &0 W323  ; Current Slab Stored Width
; rung 35
LDNOT W16.10  ; Slab Data Read in Progress
ANDNOT W16.11  ; Block Data Read in Progress
AND<>(305) W322 W323  ; Current Slab Last Width, Current Slab Stored Width
OUT W37.11  ; Last and Stored Slab Sizes are Not Equal
; rung 36
@LD W37.11  ; Last and Stored Slab Sizes are Not Equal
DIST(080) W208 DR1,IR1 &0  ; Current Slab Size in inches
; rung 37
LDNOT W16.10  ; Slab Data Read in Progress
ANDNOT W16.11  ; Block Data Read in Progress
AND<>(305) W324 W209  ; Current Slab Last Quantity, Current Slab Quantity to cut
OUT W37.12  ; Last and Current Slab Qty are Not Equal
; rung 38
@LD W37.12  ; Last and Current Slab Qty are Not Equal
MOV(021) W209 W324  ; Current Slab Quantity to cut, Current Slab Last Quantity
COLL(081) DR1,IR1 &1 W325  ; Current Slab Stored Quantity
; rung 39
LDNOT W16.10  ; Slab Data Read in Progress
ANDNOT W16.11  ; Block Data Read in Progress
AND<>(305) W324 W325  ; Current Slab Last Quantity, Current Slab Stored Quantity
OUT W37.13  ; Last and Stored Slab Qty are Not Equal

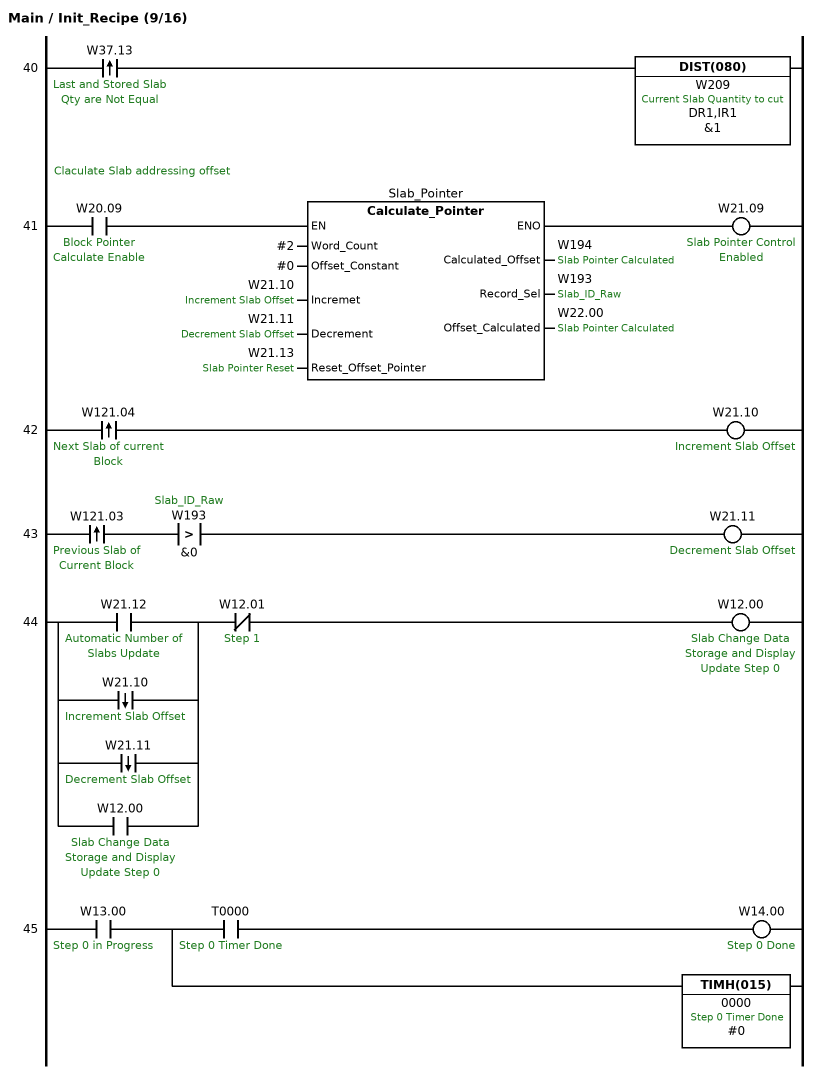
; rung 40
@LD W37.13  ; Last and Stored Slab Qty are Not Equal
DIST(080) W209 DR1,IR1 &1  ; Current Slab Quantity to cut
; rung 41: Claculate Slab addressing offset
LD W20.09  ; Block Pointer Calculate Enable
CALL Slab_Pointer : Calculate_Pointer (Word_Count := #2, Offset_Constant := #0, Incremet := W21.10, Decrement := W21.11, Reset_Offset_Pointer := W21.13, Calculated_Offset => W194, Record_Sel => W193, Offset_Calculated => W22.00)  ; Increment Slab Offset, Decrement Slab Offset, Slab Pointer Reset, Slab Pointer Calculated, Slab_ID_Raw
OUT W21.09  ; Slab Pointer Control Enabled
; rung 42
@LD W121.04  ; Next Slab of current Block
OUT W21.10  ; Increment Slab Offset
; rung 43
@LD W121.03  ; Previous Slab of Current Block
AND>(320) W193 &0  ; Slab_ID_Raw
OUT W21.11  ; Decrement Slab Offset
; rung 44
LD W21.12  ; Automatic Number of Slabs Update
%OR W21.10  ; Increment Slab Offset
%OR W21.11  ; Decrement Slab Offset
OR W12.00  ; Slab Change Data Storage and Display Update Step 0
ANDNOT W12.01  ; Step 1
OUT W12.00  ; Slab Change Data Storage and Display Update Step 0
; rung 45
LD W13.00  ; Step 0 in Progress
OUT TR0
AND T0000  ; Step 0 Timer Done
OUT W14.00  ; Step 0 Done
LD TR0
TIMH(015) 0000 #0  ; Step 0 Timer Done

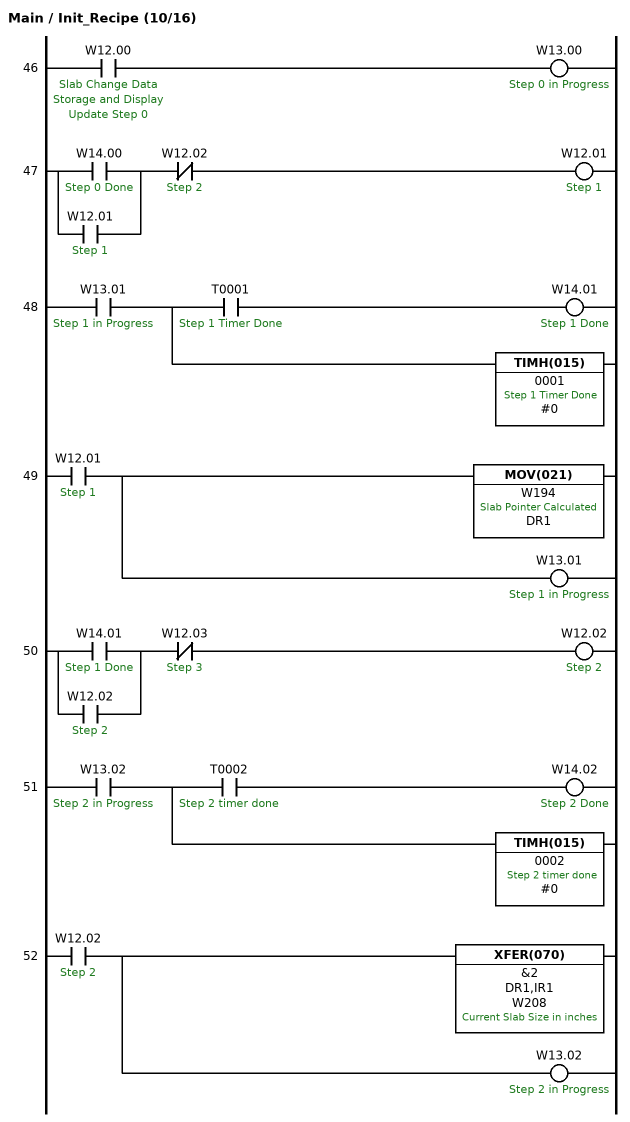
; rung 46
LD W12.00  ; Slab Change Data Storage and Display Update Step 0
OUT W13.00  ; Step 0 in Progress
; rung 47
LD W14.00  ; Step 0 Done
OR W12.01  ; Step 1
ANDNOT W12.02  ; Step 2
OUT W12.01  ; Step 1
; rung 48
LD W13.01  ; Step 1 in Progress
OUT TR0
AND T0001  ; Step 1 Timer Done
OUT W14.01  ; Step 1 Done
LD TR0
TIMH(015) 0001 #0  ; Step 1 Timer Done
; rung 49
LD W12.01  ; Step 1
MOV(021) W194 DR1  ; Slab Pointer Calculated
OUT W13.01  ; Step 1 in Progress
; rung 50
LD W14.01  ; Step 1 Done
OR W12.02  ; Step 2
ANDNOT W12.03  ; Step 3
OUT W12.02  ; Step 2
; rung 51
LD W13.02  ; Step 2 in Progress
OUT TR0
AND T0002  ; Step 2 timer done
OUT W14.02  ; Step 2 Done
LD TR0
TIMH(015) 0002 #0  ; Step 2 timer done
; rung 52
LD W12.02  ; Step 2
XFER(070) &2 DR1,IR1 W208  ; Current Slab Size in inches
OUT W13.02  ; Step 2 in Progress

